Yaskawa INFORM job: v1_150 (2).JBI

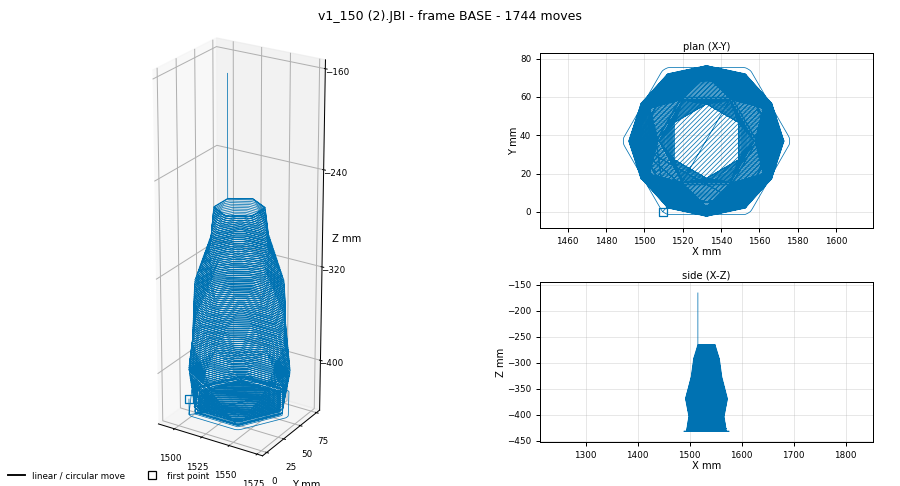
[picture p0: tool path of v1_150 (2).JBI in frame BASE, 1744 of 1745 moves have a stored position in this frame; points joined in program order, loops and branches not executed]
/JOB
//NAME v1_150
//POS
///NPOS 1745,0,0,0,0,0
///TOOL 10
///POSTYPE PULSE
///PULSE
C00000=0,15,42,180,57,90
///TOOL 10
///POSTYPE BASE
///RECTAN
///RCONF 0,0,0,0,0,0,0,0
C00001=1509.595,0.130,-417.872,180.00,-0.00,0.00
C00002=1509.595,0.130,-431.372,-180.00,-0.00,0.00
C00003=1510.195,-0.324,-431.372,180.00,-0.00,0.00
C00004=1510.690,-0.621,-431.372,180.00,-0.00,0.00
C00005=1511.242,-0.928,-431.372,180.00,-0.00,0.00
C00006=1511.746,-1.163,-431.372,-180.00,-0.00,0.00
C00007=1512.279,-1.323,-431.372,-180.00,-0.00,0.00
C00008=1513.047,-1.416,-431.372,-180.00,-0.00,0.00
C00009=1514.162,-1.438,-431.372,180.00,-0.00,0.00
C00010=1551.066,-1.438,-431.372,180.00,-0.00,0.00
C00011=1551.770,-1.428,-431.372,180.00,-0.00,0.00
C00012=1552.324,-1.380,-431.372,-180.00,-0.00,0.00
C00013=1552.866,-1.253,-431.372,-180.00,-0.00,0.00
C00014=1553.563,-0.959,-431.372,180.00,-0.00,0.00
C00015=1554.028,-0.703,-431.372,-180.00,-0.00,0.00
C00016=1554.602,-0.361,-431.372,-180.00,-0.00,0.00
C00017=1555.059,-0.043,-431.372,-180.00,-0.00,0.00
C00018=1555.465,0.338,-431.372,-180.00,-0.00,0.00
C00019=1555.933,0.960,-431.372,-180.00,-0.00,0.00
C00020=1556.527,1.941,-431.372,180.00,-0.00,0.00
///RCONF 0,0,0,1,0,0,0,0
C00021=1574.971,33.887,-431.372,180.00,-0.00,0.00
C00022=1575.305,34.482,-431.372,180.00,-0.00,0.00
C00023=1575.542,34.986,-431.372,180.00,-0.00,0.00
C00024=1575.704,35.518,-431.372,180.00,-0.00,0.00
C00025=1575.800,36.272,-431.372,180.00,-0.00,0.00
C00026=1575.812,36.838,-431.372,180.00,-0.00,0.00
C00027=1575.802,37.485,-431.372,180.00,-0.00,0.00
C00028=1575.753,38.039,-431.372,180.00,-0.00,0.00
C00029=1575.626,38.581,-431.372,-180.00,-0.00,0.00
C00030=1575.323,39.291,-431.372,-180.00,-0.00,0.00
C00031=1574.749,40.335,-431.372,-180.00,-0.00,0.00
C00032=1556.343,72.213,-431.372,180.00,-0.00,0.00
C00033=1555.982,72.818,-431.372,-180.00,-0.00,0.00
C00034=1555.663,73.274,-431.372,-180.00,-0.00,0.00
C00035=1555.282,73.679,-431.372,180.00,-0.00,0.00
C00036=1554.663,74.145,-431.372,-180.00,-0.00,0.00
C00037=1553.870,74.624,-431.372,180.00,-0.00,0.00
C00038=1553.416,74.870,-431.372,-180.00,-0.00,0.00
C00039=1553.391,74.882,-431.372,180.00,-0.00,0.00
C00040=1552.873,75.087,-431.372,180.00,-0.00,0.00
C00041=1552.332,75.214,-431.372,180.00,-0.00,0.00
C00042=1551.828,75.262,-431.372,-180.00,-0.00,0.00
C00043=1551.375,75.274,-431.372,180.00,-0.00,0.00
C00044=1513.794,75.274,-431.372,180.00,-0.00,0.00
C00045=1513.090,75.264,-431.372,-180.00,-0.00,0.00
C00046=1512.536,75.216,-431.372,180.00,-0.00,0.00
C00047=1511.994,75.089,-431.372,180.00,-0.00,0.00
C00048=1511.295,74.794,-431.372,180.00,-0.00,0.00
C00049=1510.814,74.529,-431.372,180.00,-0.00,0.00
C00050=1510.254,74.195,-431.372,-180.00,-0.00,0.00
C00051=1509.798,73.876,-431.372,-180.00,-0.00,0.00
C00052=1509.392,73.496,-431.372,-180.00,-0.00,0.00
C00053=1508.921,72.869,-431.372,-180.00,-0.00,0.00
C00054=1508.309,71.854,-431.372,180.00,-0.00,0.00
C00055=1489.889,39.948,-431.372,-180.00,-0.00,0.00
C00056=1489.554,39.351,-431.372,-180.00,-0.00,0.00
C00057=1489.317,38.848,-431.372,-180.00,-0.00,0.00
C00058=1489.155,38.315,-431.372,180.00,-0.00,0.00
C00059=1489.059,37.553,-431.372,180.00,-0.00,0.00
C00060=1489.048,36.998,-431.372,180.00,-0.00,0.00
C00061=1489.058,36.351,-431.372,180.00,-0.00,0.00
C00062=1489.107,35.797,-431.372,180.00,-0.00,0.00
C00063=1489.234,35.255,-431.372,-180.00,-0.00,0.00
C00064=1489.537,34.545,-431.372,180.00,-0.00,0.00
C00065=1490.111,33.501,-431.372,180.00,-0.00,0.00
///RCONF 0,0,0,0,0,0,0,0
C00066=1508.511,1.634,-431.372,180.00,-0.00,0.00
C00067=1508.895,0.991,-431.372,-180.00,-0.00,0.00
C00068=1509.214,0.535,-431.372,180.00,-0.00,0.00
C00069=1509.595,0.130,-431.372,-180.00,-0.00,0.00
///RCONF 0,0,0,1,0,0,0,0
C00070=1512.867,3.628,-431.372,180.00,-0.00,0.00
C00071=1551.455,70.424,-431.372,-180.00,-0.00,0.00
C00072=1551.482,70.524,-431.372,180.00,-0.00,0.00
C00073=1513.378,70.524,-431.372,-180.00,-0.00,0.00
C00074=1512.852,70.220,-431.372,180.00,-0.00,0.00
C00075=1493.798,37.220,-431.372,-180.00,-0.00,0.00
C00076=1493.799,36.615,-431.372,180.00,-0.00,0.00
C00077=1512.853,3.614,-431.372,180.00,-0.00,0.00
C00078=1513.378,3.312,-431.372,-180.00,-0.00,0.00
C00079=1551.482,3.312,-431.372,180.00,-0.00,0.00
C00080=1552.008,3.616,-431.372,-180.00,-0.00,0.00
C00081=1571.062,36.616,-431.372,-180.00,-0.00,0.00
C00082=1571.061,37.221,-431.372,180.00,-0.00,0.00
C00083=1552.008,70.220,-431.372,180.00,-0.00,0.00
C00084=1551.482,70.524,-431.372,180.00,-0.00,0.00
C00085=1550.607,70.524,-431.372,180.00,-0.00,0.00
C00086=1550.607,70.424,-431.372,180.00,-0.00,0.00
C00087=1550.827,68.784,-431.372,180.00,-0.00,0.00
C00088=1514.033,68.784,-431.372,180.00,-0.00,0.00
C00089=1495.634,36.919,-431.372,180.00,-0.00,0.00
C00090=1514.032,5.052,-431.372,180.00,-0.00,0.00
C00091=1550.827,5.052,-431.372,180.00,-0.00,0.00
C00092=1569.226,36.917,-431.372,-180.00,-0.00,0.00
C00093=1550.827,68.784,-431.372,180.00,-0.00,0.00
C00094=1516.485,67.996,-431.372,180.00,-0.00,0.00
C00095=1511.757,63.268,-431.372,-180.00,-0.00,0.00
C00096=1511.448,62.959,-431.372,-180.00,-0.00,0.00
C00097=1508.376,57.412,-431.372,180.00,-0.00,0.00
C00098=1518.960,67.996,-431.372,180.00,-0.00,0.00
C00099=1521.435,67.996,-431.372,180.00,-0.00,0.00
C00100=1504.995,51.555,-431.372,-180.00,-0.00,0.00
C00101=1504.686,51.246,-431.372,-180.00,-0.00,0.00
C00102=1501.614,45.700,-431.372,180.00,-0.00,0.00
C00103=1523.910,67.996,-431.372,-180.00,-0.00,0.00
C00104=1526.385,67.996,-431.372,-180.00,-0.00,0.00
C00105=1498.233,39.844,-431.372,180.00,-0.00,0.00
C00106=1497.924,39.535,-431.372,-180.00,-0.00,0.00
C00107=1496.995,36.131,-431.372,-180.00,-0.00,0.00
C00108=1528.859,67.996,-431.372,-180.00,-0.00,0.00
C00109=1531.334,67.996,-431.372,-180.00,-0.00,0.00
C00110=1497.901,34.562,-431.372,180.00,-0.00,0.00
C00111=1498.807,32.993,-431.372,-180.00,-0.00,0.00
C00112=1533.809,67.996,-431.372,-180.00,-0.00,0.00
C00113=1536.284,67.996,-431.372,180.00,-0.00,0.00
C00114=1499.713,31.424,-431.372,-180.00,-0.00,0.00
C00115=1500.618,29.855,-431.372,180.00,-0.00,0.00
C00116=1538.759,67.996,-431.372,-180.00,-0.00,0.00
C00117=1541.234,67.996,-431.372,180.00,-0.00,0.00
C00118=1501.524,28.286,-431.372,-180.00,-0.00,0.00
C00119=1502.430,26.717,-431.372,180.00,-0.00,0.00
C00120=1543.709,67.996,-431.372,180.00,-0.00,0.00
C00121=1546.184,67.996,-431.372,180.00,-0.00,0.00
C00122=1503.336,25.149,-431.372,180.00,-0.00,0.00
C00123=1504.242,23.579,-431.372,180.00,-0.00,0.00
C00124=1548.658,67.996,-431.372,-180.00,-0.00,0.00
C00125=1550.650,67.513,-431.372,180.00,-0.00,0.00
C00126=1505.148,22.010,-431.372,180.00,-0.00,0.00
C00127=1506.054,20.441,-431.372,180.00,-0.00,0.00
C00128=1551.556,65.944,-431.372,180.00,-0.00,0.00
C00129=1552.462,64.375,-431.372,180.00,-0.00,0.00
C00130=1506.960,18.872,-431.372,-180.00,-0.00,0.00
C00131=1507.865,17.303,-431.372,-180.00,-0.00,0.00
C00132=1553.369,62.806,-431.372,-180.00,-0.00,0.00
C00133=1554.274,61.237,-431.372,180.00,-0.00,0.00
C00134=1508.771,15.734,-431.372,180.00,-0.00,0.00
C00135=1509.677,14.165,-431.372,-180.00,-0.00,0.00
C00136=1555.180,59.668,-431.372,-180.00,-0.00,0.00
C00137=1556.086,58.099,-431.372,180.00,-0.00,0.00
C00138=1510.583,12.596,-431.372,180.00,-0.00,0.00
C00139=1511.489,11.027,-431.372,-180.00,-0.00,0.00
C00140=1556.992,56.530,-431.372,-180.00,-0.00,0.00
C00141=1557.898,54.961,-431.372,180.00,-0.00,0.00
C00142=1512.394,9.458,-431.372,-180.00,-0.00,0.00
C00143=1513.300,7.889,-431.372,-180.00,-0.00,0.00
C00144=1558.804,53.393,-431.372,-180.00,-0.00,0.00
C00145=1559.710,51.823,-431.372,180.00,-0.00,0.00
C00146=1514.206,6.320,-431.372,-180.00,-0.00,0.00
C00147=1516.200,5.839,-431.372,-180.00,-0.00,0.00
C00148=1560.616,50.254,-431.372,-180.00,-0.00,0.00
C00149=1561.521,48.685,-431.372,-180.00,-0.00,0.00
C00150=1518.675,5.839,-431.372,-180.00,-0.00,0.00
C00151=1521.150,5.839,-431.372,-180.00,-0.00,0.00
C00152=1562.427,47.116,-431.372,180.00,-0.00,0.00
C00153=1563.333,45.547,-431.372,180.00,-0.00,0.00
C00154=1523.625,5.839,-431.372,-180.00,-0.00,0.00
C00155=1526.100,5.839,-431.372,-180.00,-0.00,0.00
C00156=1564.240,43.979,-431.372,180.00,-0.00,0.00
C00157=1565.145,42.410,-431.372,180.00,-0.00,0.00
C00158=1528.575,5.839,-431.372,-180.00,-0.00,0.00
C00159=1531.049,5.839,-431.372,-180.00,-0.00,0.00
C00160=1566.051,40.841,-431.372,-180.00,-0.00,0.00
C00161=1566.957,39.272,-431.372,180.00,-0.00,0.00
C00162=1533.524,5.839,-431.372,180.00,-0.00,0.00
C00163=1535.999,5.839,-431.372,-180.00,-0.00,0.00
C00164=1567.863,37.703,-431.372,-180.00,-0.00,0.00
C00165=1568.172,38.012,-431.372,180.00,-0.00,0.00
C00166=1566.627,33.992,-431.372,-180.00,-0.00,0.00
C00167=1538.474,5.839,-431.372,-180.00,-0.00,0.00
C00168=1540.949,5.839,-431.372,-180.00,-0.00,0.00
C00169=1563.246,28.136,-431.372,-180.00,-0.00,0.00
C00170=1563.555,28.445,-431.372,180.00,-0.00,0.00
C00171=1559.865,22.280,-431.372,180.00,-0.00,0.00
C00172=1543.424,5.839,-431.372,180.00,-0.00,0.00
C00173=1545.899,5.839,-431.372,180.00,-0.00,0.00
C00174=1556.483,16.424,-431.372,180.00,-0.00,0.00
C00175=1556.792,16.733,-431.372,180.00,-0.00,0.00
C00176=1553.102,10.567,-431.372,-180.00,-0.00,0.00
C00177=1548.373,5.839,-431.372,180.00,-0.00,0.00
C00178=1548.064,5.530,-431.372,-180.00,-0.00,0.00
C00179=1548.064,5.530,-429.872,-180.00,-0.00,0.00
C00180=1494.414,35.749,-429.872,-180.00,-0.00,0.00
C00181=1494.043,35.534,-429.872,180.00,-0.00,0.00
C00182=1512.039,4.366,-429.872,180.00,-0.00,0.00
C00183=1514.436,2.983,-429.872,180.00,-0.00,0.00
C00184=1550.425,2.983,-429.872,180.00,-0.00,0.00
C00185=1552.822,4.368,-429.872,180.00,-0.00,0.00
C00186=1570.817,35.535,-429.872,-180.00,-0.00,0.00
C00187=1570.817,38.302,-429.872,-180.00,-0.00,0.00
C00188=1552.821,69.470,-429.872,-180.00,-0.00,0.00
C00189=1550.424,70.853,-429.872,180.00,-0.00,0.00
C00190=1514.435,70.853,-429.872,180.00,-0.00,0.00
C00191=1512.038,69.468,-429.872,-180.00,-0.00,0.00
C00192=1494.043,38.301,-429.872,180.00,-0.00,0.00
C00193=1494.043,35.534,-429.872,180.00,-0.00,0.00
C00194=1493.799,36.615,-429.872,180.00,-0.00,0.00
C00195=1512.278,4.505,-429.633,-180.00,-0.00,0.00
C00196=1514.436,3.256,-429.617,180.00,-0.00,0.00
C00197=1550.425,3.206,-429.385,180.00,-0.00,0.00
C00198=1552.632,4.477,-429.369,180.00,-0.00,0.00
C00199=1570.671,35.619,-429.137,-180.00,-0.00,0.00
C00200=1570.675,38.219,-429.120,-180.00,-0.00,0.00
C00201=1552.723,69.413,-428.888,-180.00,-0.00,0.00
C00202=1550.424,70.743,-428.871,180.00,-0.00,0.00
C00203=1514.435,70.794,-428.639,-180.00,-0.00,0.00
C00204=1512.086,69.440,-428.622,-180.00,-0.00,0.00
C00205=1494.047,38.299,-428.390,-180.00,-0.00,0.00
C00206=1494.043,35.534,-428.372,-180.00,-0.00,0.00
C00207=1519.293,14.162,-428.070,-180.00,-0.00,0.00
C00208=1545.567,14.162,-427.831,180.00,-0.00,0.00
C00209=1558.706,36.918,-427.591,180.00,-0.00,0.00
C00210=1545.567,59.674,-427.351,180.00,-0.00,0.00
C00211=1519.293,59.674,-427.112,-180.00,-0.00,0.00
C00212=1506.154,36.918,-426.872,180.00,-0.00,0.00
C00213=1506.266,36.912,-426.872,180.00,-0.00,0.00
C00214=1519.303,59.657,-426.872,-180.00,-0.00,0.00
C00215=1517.955,60.437,-426.872,180.00,-0.00,0.00
C00216=1512.921,63.340,-426.872,180.00,-0.00,0.00
C00217=1511.588,64.111,-426.872,-180.00,-0.00,0.00
C00218=1513.794,68.122,-426.872,-180.00,-0.00,0.00
C00219=1513.864,68.052,-426.872,-180.00,-0.00,0.00
C00220=1514.750,68.563,-426.872,-180.00,-0.00,0.00
C00221=1550.109,68.564,-426.872,-180.00,-0.00,0.00
C00222=1550.995,68.053,-426.872,-180.00,-0.00,0.00
C00223=1568.676,37.431,-426.872,180.00,-0.00,0.00
C00224=1568.677,36.407,-426.872,-180.00,-0.00,0.00
C00225=1550.996,5.784,-426.872,180.00,-0.00,0.00
C00226=1550.110,5.273,-426.872,-180.00,-0.00,0.00
C00227=1514.751,5.272,-426.872,180.00,-0.00,0.00
C00228=1513.865,5.783,-426.872,-180.00,-0.00,0.00
C00229=1496.184,36.405,-426.872,-180.00,-0.00,0.00
C00230=1496.183,37.429,-426.872,-180.00,-0.00,0.00
C00231=1513.864,68.052,-426.872,-180.00,-0.00,0.00
C00232=1514.622,68.489,-426.872,-180.00,-0.00,0.00
C00233=1514.571,68.575,-426.872,-180.00,-0.00,0.00
C00234=1549.340,71.086,-426.872,-180.00,-0.00,0.00
C00235=1549.365,71.182,-426.872,180.00,-0.00,0.00
C00236=1515.494,71.182,-426.872,-180.00,-0.00,0.00
C00237=1511.223,68.715,-426.872,180.00,-0.00,0.00
C00238=1494.287,39.382,-426.872,-180.00,-0.00,0.00
C00239=1494.288,34.451,-426.872,180.00,-0.00,0.00
C00240=1511.225,5.118,-426.872,-180.00,-0.00,0.00
C00241=1515.495,2.654,-426.872,180.00,-0.00,0.00
C00242=1549.366,2.654,-426.872,-180.00,-0.00,0.00
C00243=1553.637,5.121,-426.872,-180.00,-0.00,0.00
C00244=1570.573,34.454,-426.872,180.00,-0.00,0.00
C00245=1570.572,39.385,-426.872,180.00,-0.00,0.00
C00246=1553.635,68.718,-426.872,-180.00,-0.00,0.00
C00247=1549.365,71.182,-426.872,180.00,-0.00,0.00
C00248=1548.490,71.182,-426.872,-180.00,-0.00,0.00
C00249=1548.490,71.082,-426.872,-180.00,-0.00,0.00
C00250=1514.750,68.563,-426.872,-180.00,-0.00,0.00
C00251=1515.160,67.025,-426.872,-180.00,-0.00,0.00
C00252=1519.303,61.214,-426.872,180.00,-0.00,0.00
C00253=1519.303,59.657,-426.872,-180.00,-0.00,0.00
C00254=1506.266,36.912,-426.872,180.00,-0.00,0.00
C00255=1506.154,36.918,-426.872,180.00,-0.00,0.00
C00256=1510.409,5.871,-426.670,-180.00,-0.00,0.00
///RCONF 0,0,0,0,0,0,0,0
C00257=1516.555,2.324,-426.624,180.00,-0.00,0.00
C00258=1548.305,2.324,-426.420,180.00,-0.00,0.00
///RCONF 0,0,0,1,0,0,0,0
C00259=1554.452,5.872,-426.374,180.00,-0.00,0.00
C00260=1570.328,33.372,-426.169,-180.00,-0.00,0.00
C00261=1570.327,40.467,-426.123,180.00,-0.00,0.00
C00262=1554.450,67.965,-425.919,180.00,-0.00,0.00
C00263=1548.305,71.512,-425.873,-180.00,-0.00,0.00
C00264=1516.555,71.512,-425.668,180.00,-0.00,0.00
C00265=1510.408,67.964,-425.622,-180.00,-0.00,0.00
C00266=1494.532,40.464,-425.418,180.00,-0.00,0.00
C00267=1494.533,33.369,-425.372,-180.00,-0.00,0.00
C00268=1509.843,6.766,-425.175,180.00,-0.00,0.00
///RCONF 0,0,0,0,0,0,0,0
C00269=1517.615,2.268,-425.117,-180.00,-0.00,0.00
C00270=1547.247,2.227,-424.927,-180.00,-0.00,0.00
///RCONF 0,0,0,1,0,0,0,0
C00271=1555.078,6.736,-424.869,180.00,-0.00,0.00
C00272=1569.930,32.380,-424.679,-180.00,-0.00,0.00
C00273=1569.942,41.464,-424.620,180.00,-0.00,0.00
C00274=1555.159,67.150,-424.430,-180.00,-0.00,0.00
C00275=1547.245,71.731,-424.371,180.00,-0.00,0.00
C00276=1517.613,71.773,-424.181,-180.00,-0.00,0.00
C00277=1509.640,67.181,-424.122,180.00,-0.00,0.00
C00278=1494.788,41.539,-423.931,-180.00,-0.00,0.00
C00279=1494.776,32.289,-423.872,180.00,-0.00,0.00
C00280=1509.032,7.522,-423.689,180.00,-0.00,0.00
///RCONF 0,0,0,0,0,0,0,0
C00281=1518.674,1.939,-423.617,180.00,-0.00,0.00
C00282=1546.188,1.901,-423.441,180.00,-0.00,0.00
///RCONF 0,0,0,1,0,0,0,0
C00283=1555.893,7.489,-423.369,-180.00,-0.00,0.00
C00284=1569.682,31.298,-423.192,-180.00,-0.00,0.00
C00285=1569.697,42.546,-423.120,-180.00,-0.00,0.00
C00286=1555.971,66.397,-422.944,-180.00,-0.00,0.00
C00287=1546.186,72.060,-422.871,180.00,-0.00,0.00
C00288=1518.672,72.099,-422.695,180.00,-0.00,0.00
C00289=1508.825,66.428,-422.622,180.00,-0.00,0.00
C00290=1495.035,42.618,-422.445,180.00,-0.00,0.00
C00291=1495.021,31.207,-422.372,180.00,-0.00,0.00
C00292=1508.218,8.276,-422.202,180.00,-0.00,0.00
///RCONF 0,0,0,0,0,0,0,0
C00293=1519.730,1.610,-422.117,180.00,-0.00,0.00
C00294=1545.130,1.575,-421.954,180.00,-0.00,0.00
///RCONF 0,0,0,1,0,0,0,0
C00295=1556.705,8.239,-421.869,180.00,-0.00,0.00
C00296=1569.436,30.219,-421.706,-180.00,-0.00,0.00
C00297=1569.452,43.627,-421.620,180.00,-0.00,0.00
C00298=1556.783,65.642,-421.457,180.00,-0.00,0.00
C00299=1545.130,72.389,-421.371,-180.00,-0.00,0.00
C00300=1519.730,72.425,-421.208,-180.00,-0.00,0.00
C00301=1508.013,65.679,-421.122,180.00,-0.00,0.00
C00302=1495.282,43.699,-420.959,180.00,-0.00,0.00
C00303=1495.266,30.126,-420.872,180.00,-0.00,0.00
C00304=1507.406,9.031,-420.716,-180.00,-0.00,0.00
///RCONF 0,0,0,0,0,0,0,0
C00305=1520.790,1.281,-420.617,-180.00,-0.00,0.00
C00306=1544.070,1.249,-420.468,-180.00,-0.00,0.00
///RCONF 0,0,0,1,0,0,0,0
C00307=1557.520,8.992,-420.369,180.00,-0.00,0.00
C00308=1569.189,29.140,-420.220,-180.00,-0.00,0.00
C00309=1569.208,44.709,-420.120,-180.00,-0.00,0.00
C00310=1557.595,64.887,-419.971,-180.00,-0.00,0.00
C00311=1544.070,72.718,-419.871,180.00,-0.00,0.00
C00312=1520.790,72.751,-419.722,180.00,-0.00,0.00
C00313=1507.199,64.925,-419.622,-180.00,-0.00,0.00
C00314=1495.530,44.781,-419.473,180.00,-0.00,0.00
C00315=1495.510,29.044,-419.372,180.00,-0.00,0.00
C00316=1506.595,9.785,-419.230,-180.00,-0.00,0.00
///RCONF 0,0,0,0,0,0,0,0
C00317=1521.848,0.952,-419.117,180.00,-0.00,0.00
C00318=1543.012,0.923,-418.982,-180.00,-0.00,0.00
///RCONF 0,0,0,1,0,0,0,0
C00319=1558.334,9.744,-418.869,-180.00,-0.00,0.00
C00320=1568.940,28.059,-418.734,180.00,-0.00,0.00
C00321=1568.963,45.792,-418.620,180.00,-0.00,0.00
C00322=1558.407,64.133,-418.485,180.00,-0.00,0.00
C00323=1543.012,73.047,-418.371,-180.00,-0.00,0.00
C00324=1521.848,73.077,-418.236,180.00,-0.00,0.00
C00325=1506.384,64.173,-418.122,180.00,-0.00,0.00
C00326=1495.777,45.861,-417.986,-180.00,-0.00,0.00
C00327=1495.755,27.961,-417.872,180.00,-0.00,0.00
C00328=1505.782,10.538,-417.744,180.00,-0.00,0.00
///RCONF 0,0,0,0,0,0,0,0
C00329=1522.907,0.623,-417.617,-180.00,-0.00,0.00
C00330=1541.953,0.597,-417.496,-180.00,-0.00,0.00
///RCONF 0,0,0,1,0,0,0,0
C00331=1559.148,10.496,-417.369,180.00,-0.00,0.00
C00332=1568.693,26.977,-417.247,180.00,-0.00,0.00
C00333=1568.719,46.873,-417.120,-180.00,-0.00,0.00
C00334=1559.219,63.380,-416.999,180.00,-0.00,0.00
C00335=1541.953,73.376,-416.871,180.00,-0.00,0.00
C00336=1522.907,73.403,-416.750,-180.00,-0.00,0.00
C00337=1505.570,63.421,-416.622,-180.00,-0.00,0.00
C00338=1496.024,46.942,-416.500,180.00,-0.00,0.00
C00339=1495.999,26.880,-416.372,180.00,-0.00,0.00
C00340=1504.971,11.292,-416.257,-180.00,-0.00,0.00
///RCONF 0,0,0,0,0,0,0,0
C00341=1523.967,0.294,-416.117,180.00,-0.00,0.00
C00342=1540.889,0.270,-416.009,-180.00,-0.00,0.00
///RCONF 0,0,0,1,0,0,0,0
C00343=1559.963,11.249,-415.869,-180.00,-0.00,0.00
C00344=1568.447,25.896,-415.761,180.00,-0.00,0.00
C00345=1568.474,47.955,-415.620,180.00,-0.00,0.00
C00346=1560.031,62.626,-415.512,-180.00,-0.00,0.00
C00347=1540.893,73.705,-415.371,-180.00,-0.00,0.00
C00348=1523.971,73.730,-415.263,-180.00,-0.00,0.00
C00349=1504.755,62.668,-415.122,180.00,-0.00,0.00
C00350=1496.271,48.022,-415.014,-180.00,-0.00,0.00
C00351=1496.244,25.798,-414.872,-180.00,-0.00,0.00
C00352=1504.158,12.046,-414.771,180.00,-0.00,0.00
///RCONF 0,0,0,0,0,0,0,0
C00353=1525.026,-0.035,-414.617,180.00,-0.00,0.00
C00354=1539.831,-0.056,-414.523,-180.00,-0.00,0.00
///RCONF 0,0,0,1,0,0,0,0
C00355=1560.777,12.001,-414.369,-180.00,-0.00,0.00
C00356=1568.200,24.816,-414.275,-180.00,-0.00,0.00
C00357=1568.230,49.036,-414.120,180.00,-0.00,0.00
C00358=1560.843,61.872,-414.026,-180.00,-0.00,0.00
C00359=1539.834,74.034,-413.871,-180.00,-0.00,0.00
C00360=1525.029,74.057,-413.777,-180.00,-0.00,0.00
C00361=1503.941,61.916,-413.622,180.00,-0.00,0.00
C00362=1496.518,49.102,-413.527,180.00,-0.00,0.00
C00363=1496.488,24.717,-413.372,-180.00,-0.00,0.00
C00364=1503.347,12.801,-413.284,-180.00,-0.00,0.00
///RCONF 0,0,0,0,0,0,0,0
C00365=1526.085,-0.364,-413.117,180.00,-0.00,0.00
C00366=1538.773,-0.382,-413.036,-180.00,-0.00,0.00
///RCONF 0,0,0,1,0,0,0,0
C00367=1561.592,12.754,-412.869,180.00,-0.00,0.00
C00368=1567.953,23.736,-412.788,180.00,-0.00,0.00
C00369=1567.985,50.118,-412.620,180.00,-0.00,0.00
C00370=1561.655,61.117,-412.539,-180.00,-0.00,0.00
C00371=1538.775,74.363,-412.371,180.00,-0.00,0.00
C00372=1526.087,74.383,-412.290,-180.00,-0.00,0.00
C00373=1503.126,61.163,-412.122,180.00,-0.00,0.00
C00374=1496.766,50.182,-412.041,-180.00,-0.00,0.00
C00375=1496.733,23.635,-411.872,180.00,-0.00,0.00
C00376=1502.535,13.554,-411.798,-180.00,-0.00,0.00
///RCONF 0,0,0,0,0,0,0,0
C00377=1527.144,-0.693,-411.617,-180.00,-0.00,0.00
C00378=1537.712,-0.708,-411.550,-180.00,-0.00,0.00
///RCONF 0,0,0,1,0,0,0,0
C00379=1562.406,13.507,-411.369,180.00,-0.00,0.00
C00380=1567.706,22.658,-411.302,180.00,-0.00,0.00
C00381=1567.740,51.200,-411.120,-180.00,-0.00,0.00
C00382=1562.467,60.364,-411.053,180.00,-0.00,0.00
C00383=1537.716,74.692,-410.871,180.00,-0.00,0.00
C00384=1527.148,74.709,-410.804,180.00,-0.00,0.00
C00385=1502.312,60.411,-410.622,-180.00,-0.00,0.00
C00386=1497.012,51.263,-410.555,180.00,-0.00,0.00
C00387=1496.978,22.553,-410.372,180.00,-0.00,0.00
C00388=1501.722,14.310,-410.312,-180.00,-0.00,0.00
///RCONF 0,0,0,0,0,0,0,0
C00389=1528.203,-1.022,-410.117,180.00,-0.00,0.00
C00390=1536.657,-1.034,-410.064,-180.00,-0.00,0.00
///RCONF 0,0,0,1,0,0,0,0
C00391=1563.221,14.259,-409.869,180.00,-0.00,0.00
C00392=1567.458,21.576,-409.815,180.00,-0.00,0.00
C00393=1567.496,52.282,-409.620,180.00,-0.00,0.00
C00394=1563.279,59.608,-409.567,180.00,-0.00,0.00
C00395=1536.657,75.022,-409.371,-180.00,-0.00,0.00
C00396=1528.203,75.034,-409.317,-180.00,-0.00,0.00
C00397=1501.497,59.657,-409.122,180.00,-0.00,0.00
C00398=1497.260,52.343,-409.068,180.00,-0.00,0.00
C00399=1497.222,21.471,-408.872,-180.00,-0.00,0.00
C00400=1500.911,15.063,-408.825,-180.00,-0.00,0.00
///RCONF 0,0,0,0,0,0,0,0
C00401=1529.262,-1.352,-408.617,180.00,-0.00,0.00
C00402=1535.598,-1.360,-408.577,180.00,-0.00,0.00
///RCONF 0,0,0,1,0,0,0,0
C00403=1564.035,15.011,-408.369,-180.00,-0.00,0.00
C00404=1567.211,20.497,-408.329,180.00,-0.00,0.00
C00405=1567.251,53.364,-408.120,-180.00,-0.00,0.00
C00406=1564.091,58.855,-408.080,-180.00,-0.00,0.00
C00407=1535.598,75.351,-407.871,180.00,-0.00,0.00
C00408=1529.262,75.360,-407.831,-180.00,-0.00,0.00
C00409=1500.683,58.906,-407.622,-180.00,-0.00,0.00
C00410=1497.506,53.423,-407.582,180.00,-0.00,0.00
C00411=1497.467,20.389,-407.372,180.00,-0.00,0.00
C00412=1500.098,15.817,-407.339,180.00,-0.00,0.00
///RCONF 0,0,0,0,0,0,0,0
C00413=1530.321,-1.681,-407.117,180.00,-0.00,0.00
C00414=1534.539,-1.686,-407.091,-180.00,-0.00,0.00
///RCONF 0,0,0,1,0,0,0,0
C00415=1564.850,15.764,-406.869,180.00,-0.00,0.00
C00416=1566.964,19.415,-406.842,180.00,-0.00,0.00
C00417=1567.007,54.445,-406.620,-180.00,-0.00,0.00
C00418=1564.903,58.101,-406.593,-180.00,-0.00,0.00
C00419=1534.539,75.680,-406.371,-180.00,-0.00,0.00
C00420=1530.321,75.686,-406.344,180.00,-0.00,0.00
C00421=1499.868,58.153,-406.122,-180.00,-0.00,0.00
C00422=1497.754,54.503,-406.095,-180.00,-0.00,0.00
C00423=1497.711,19.308,-405.872,180.00,-0.00,0.00
C00424=1499.287,16.571,-405.852,180.00,-0.00,0.00
///RCONF 0,0,0,0,0,0,0,0
C00425=1531.380,-2.010,-405.617,-180.00,-0.00,0.00
C00426=1533.480,-2.012,-405.604,180.00,-0.00,0.00
///RCONF 0,0,0,1,0,0,0,0
C00427=1565.665,16.517,-405.369,-180.00,-0.00,0.00
C00428=1566.718,18.336,-405.356,180.00,-0.00,0.00
C00429=1566.762,55.528,-405.120,-180.00,-0.00,0.00
C00430=1565.715,57.347,-405.107,180.00,-0.00,0.00
C00431=1533.480,76.009,-404.871,-180.00,-0.00,0.00
C00432=1531.380,76.012,-404.858,180.00,-0.00,0.00
C00433=1499.053,57.400,-404.622,180.00,-0.00,0.00
C00434=1498.000,55.582,-404.608,-180.00,-0.00,0.00
C00435=1497.956,18.225,-404.372,180.00,-0.00,0.00
///RCONF 0,0,0,0,0,0,0,0
C00436=1532.430,-2.337,-404.118,-180.00,-0.00,0.00
///RCONF 0,0,0,1,0,0,0,0
C00437=1566.473,17.262,-403.870,180.00,-0.00,0.00
C00438=1566.520,56.600,-403.621,180.00,-0.00,0.00
C00439=1532.430,76.335,-403.371,-180.00,-0.00,0.00
C00440=1498.247,56.654,-403.122,180.00,-0.00,0.00
C00441=1498.200,17.155,-402.872,-180.00,-0.00,0.00
C00442=1498.701,16.866,-402.868,-180.00,-0.00,0.00
///RCONF 0,0,0,0,0,0,0,0
C00443=1531.912,-2.345,-402.625,-180.00,-0.00,0.00
C00444=1532.946,-2.348,-402.618,-180.00,-0.00,0.00
///RCONF 0,0,0,1,0,0,0,0
C00445=1566.189,16.806,-402.375,-180.00,-0.00,0.00
C00446=1566.728,17.735,-402.368,180.00,-0.00,0.00
C00447=1566.761,56.103,-402.124,-180.00,-0.00,0.00
C00448=1566.210,57.059,-402.117,180.00,-0.00,0.00
C00449=1532.999,76.270,-401.874,180.00,-0.00,0.00
C00450=1531.863,76.273,-401.867,180.00,-0.00,0.00
C00451=1498.620,57.118,-401.623,180.00,-0.00,0.00
C00452=1498.030,56.101,-401.616,-180.00,-0.00,0.00
C00453=1497.997,17.732,-401.372,-180.00,-0.00,0.00
C00454=1499.367,16.243,-401.359,-180.00,-0.00,0.00
///RCONF 0,0,0,0,0,0,0,0
C00455=1531.037,-2.090,-401.127,180.00,-0.00,0.00
C00456=1533.826,-2.093,-401.109,180.00,-0.00,0.00
///RCONF 0,0,0,1,0,0,0,0
C00457=1565.541,16.165,-400.876,-180.00,-0.00,0.00
C00458=1566.961,18.619,-400.858,180.00,-0.00,0.00
C00459=1567.005,55.219,-400.626,-180.00,-0.00,0.00
C00460=1565.566,57.716,-400.607,-180.00,-0.00,0.00
C00461=1533.895,76.052,-400.375,180.00,-0.00,0.00
C00462=1530.962,76.054,-400.356,-180.00,-0.00,0.00
C00463=1499.247,57.795,-400.124,180.00,-0.00,0.00
C00464=1497.755,55.217,-400.105,180.00,-0.00,0.00
C00465=1497.711,18.619,-399.872,180.00,-0.00,0.00
C00466=1499.988,15.552,-399.848,-180.00,-0.00,0.00
///RCONF 0,0,0,0,0,0,0,0
C00467=1530.127,-1.897,-399.627,180.00,-0.00,0.00
C00468=1534.738,-1.900,-399.597,180.00,-0.00,0.00
///RCONF 0,0,0,1,0,0,0,0
C00469=1564.918,15.475,-399.376,180.00,-0.00,0.00
C00470=1567.250,19.504,-399.347,-180.00,-0.00,0.00
C00471=1567.292,54.331,-399.126,180.00,-0.00,0.00
C00472=1564.944,58.409,-399.096,-180.00,-0.00,0.00
C00473=1534.805,75.858,-398.875,-180.00,-0.00,0.00
C00474=1530.050,75.861,-398.845,-180.00,-0.00,0.00
C00475=1499.870,58.485,-398.624,180.00,-0.00,0.00
C00476=1497.466,54.332,-398.593,-180.00,-0.00,0.00
C00477=1497.424,19.504,-398.372,-180.00,-0.00,0.00
C00478=1500.611,14.858,-398.336,180.00,-0.00,0.00
///RCONF 0,0,0,0,0,0,0,0
C00479=1529.216,-1.701,-398.127,-180.00,-0.00,0.00
C00480=1535.650,-1.708,-398.086,-180.00,-0.00,0.00
///RCONF 0,0,0,1,0,0,0,0
C00481=1564.293,14.783,-397.876,180.00,-0.00,0.00
C00482=1567.539,20.391,-397.835,-180.00,-0.00,0.00
C00483=1567.579,53.443,-397.626,180.00,-0.00,0.00
C00484=1564.320,59.103,-397.584,180.00,-0.00,0.00
C00485=1535.716,75.662,-397.375,180.00,-0.00,0.00
C00486=1529.138,75.668,-397.333,-180.00,-0.00,0.00
C00487=1500.495,59.177,-397.124,-180.00,-0.00,0.00
C00488=1497.176,53.445,-397.082,180.00,-0.00,0.00
C00489=1497.137,20.391,-396.872,180.00,-0.00,0.00
C00490=1501.234,14.167,-396.825,180.00,-0.00,0.00
///RCONF 0,0,0,0,0,0,0,0
C00491=1528.303,-1.505,-396.627,180.00,-0.00,0.00
C00492=1536.559,-1.517,-396.574,-180.00,-0.00,0.00
///RCONF 0,0,0,1,0,0,0,0
C00493=1563.669,14.092,-396.376,-180.00,-0.00,0.00
C00494=1567.828,21.277,-396.324,180.00,-0.00,0.00
C00495=1567.865,52.558,-396.126,180.00,-0.00,0.00
C00496=1563.698,59.795,-396.073,180.00,-0.00,0.00
C00497=1536.629,75.466,-395.875,-180.00,-0.00,0.00
C00498=1528.229,75.477,-395.822,-180.00,-0.00,0.00
C00499=1501.119,59.868,-395.624,180.00,-0.00,0.00
C00500=1496.888,52.559,-395.570,-180.00,-0.00,0.00
C00501=1496.851,21.277,-395.372,180.00,-0.00,0.00
C00502=1501.857,13.474,-395.313,180.00,-0.00,0.00
///RCONF 0,0,0,0,0,0,0,0
C00503=1527.395,-1.312,-395.127,180.00,-0.00,0.00
C00504=1537.472,-1.323,-395.063,180.00,-0.00,0.00
///RCONF 0,0,0,1,0,0,0,0
C00505=1563.044,13.400,-394.876,-180.00,-0.00,0.00
C00506=1568.117,22.163,-394.812,-180.00,-0.00,0.00
C00507=1568.152,51.672,-394.626,-180.00,-0.00,0.00
C00508=1563.075,60.487,-394.561,-180.00,-0.00,0.00
C00509=1537.537,75.273,-394.375,180.00,-0.00,0.00
C00510=1527.315,75.283,-394.310,-180.00,-0.00,0.00
C00511=1501.744,60.561,-394.124,-180.00,-0.00,0.00
C00512=1496.599,51.673,-394.059,180.00,-0.00,0.00
C00513=1496.564,22.163,-393.872,180.00,-0.00,0.00
C00514=1502.481,12.780,-393.802,180.00,-0.00,0.00
///RCONF 0,0,0,0,0,0,0,0
C00515=1526.483,-1.117,-393.627,-180.00,-0.00,0.00
C00516=1538.384,-1.130,-393.552,180.00,-0.00,0.00
///RCONF 0,0,0,1,0,0,0,0
C00517=1562.420,12.708,-393.376,180.00,-0.00,0.00
C00518=1568.406,23.051,-393.301,180.00,-0.00,0.00
C00519=1568.439,50.786,-393.126,-180.00,-0.00,0.00
C00520=1562.451,61.181,-393.050,-180.00,-0.00,0.00
C00521=1538.449,75.078,-392.875,-180.00,-0.00,0.00
C00522=1526.403,75.090,-392.799,-180.00,-0.00,0.00
C00523=1502.368,61.252,-392.624,-180.00,-0.00,0.00
C00524=1496.310,50.785,-392.547,-180.00,-0.00,0.00
C00525=1496.277,23.049,-392.372,180.00,-0.00,0.00
C00526=1503.104,12.087,-392.291,-180.00,-0.00,0.00
///RCONF 0,0,0,0,0,0,0,0
C00527=1525.573,-0.923,-392.127,180.00,-0.00,0.00
C00528=1539.295,-0.937,-392.040,180.00,-0.00,0.00
///RCONF 0,0,0,1,0,0,0,0
C00529=1561.797,12.018,-391.876,-180.00,-0.00,0.00
C00530=1568.695,23.935,-391.790,180.00,-0.00,0.00
C00531=1568.726,49.896,-391.626,-180.00,-0.00,0.00
C00532=1561.828,61.874,-391.539,-180.00,-0.00,0.00
C00533=1539.359,74.884,-391.375,-180.00,-0.00,0.00
C00534=1525.492,74.897,-391.287,180.00,-0.00,0.00
C00535=1502.991,61.942,-391.124,-180.00,-0.00,0.00
C00536=1496.022,49.901,-391.036,180.00,-0.00,0.00
C00537=1495.989,23.939,-390.872,180.00,-0.00,0.00
C00538=1503.727,11.394,-390.779,180.00,-0.00,0.00
///RCONF 0,0,0,0,0,0,0,0
C00539=1524.662,-0.727,-390.627,-180.00,-0.00,0.00
C00540=1540.208,-0.743,-390.529,180.00,-0.00,0.00
///RCONF 0,0,0,1,0,0,0,0
C00541=1561.171,11.326,-390.376,-180.00,-0.00,0.00
C00542=1568.983,24.825,-390.278,180.00,-0.00,0.00
C00543=1569.012,49.015,-390.126,180.00,-0.00,0.00
C00544=1561.205,62.567,-390.027,-180.00,-0.00,0.00
C00545=1540.270,74.688,-389.875,-180.00,-0.00,0.00
C00546=1524.580,74.704,-389.776,180.00,-0.00,0.00
C00547=1503.617,62.636,-389.624,-180.00,-0.00,0.00
C00548=1495.733,49.011,-389.524,-180.00,-0.00,0.00
C00549=1495.704,24.821,-389.372,-180.00,-0.00,0.00
C00550=1504.350,10.700,-389.268,-180.00,-0.00,0.00
///RCONF 0,0,0,0,0,0,0,0
C00551=1523.751,-0.532,-389.127,180.00,-0.00,0.00
C00552=1541.120,-0.550,-389.017,-180.00,-0.00,0.00
///RCONF 0,0,0,1,0,0,0,0
C00553=1560.548,10.634,-388.876,180.00,-0.00,0.00
C00554=1569.273,25.708,-388.767,180.00,-0.00,0.00
C00555=1569.299,48.127,-388.626,-180.00,-0.00,0.00
C00556=1560.582,63.261,-388.516,180.00,-0.00,0.00
C00557=1541.181,74.493,-388.375,180.00,-0.00,0.00
C00558=1523.668,74.511,-388.265,-180.00,-0.00,0.00
C00559=1504.240,63.326,-388.124,180.00,-0.00,0.00
C00560=1495.443,48.128,-388.013,180.00,-0.00,0.00
C00561=1495.417,25.708,-387.872,-180.00,-0.00,0.00
C00562=1504.972,10.007,-387.756,180.00,-0.00,0.00
///RCONF 0,0,0,0,0,0,0,0
C00563=1522.838,-0.336,-387.627,-180.00,-0.00,0.00
C00564=1542.032,-0.358,-387.506,-180.00,-0.00,0.00
///RCONF 0,0,0,1,0,0,0,0
C00565=1559.923,9.942,-387.376,-180.00,-0.00,0.00
C00566=1569.561,26.594,-387.255,-180.00,-0.00,0.00
C00567=1569.586,47.237,-387.126,180.00,-0.00,0.00
C00568=1559.959,63.954,-387.005,-180.00,-0.00,0.00
C00569=1542.094,74.297,-386.875,180.00,-0.00,0.00
C00570=1522.756,74.319,-386.753,180.00,-0.00,0.00
C00571=1504.865,64.018,-386.624,180.00,-0.00,0.00
C00572=1495.155,47.242,-386.502,180.00,-0.00,0.00
C00573=1495.129,26.598,-386.372,-180.00,-0.00,0.00
C00574=1505.595,9.313,-386.245,-180.00,-0.00,0.00
///RCONF 0,0,0,0,0,0,0,0
C00575=1521.931,-0.144,-386.127,-180.00,-0.00,0.00
C00576=1542.943,-0.166,-385.995,180.00,-0.00,0.00
///RCONF 0,0,0,1,0,0,0,0
C00577=1559.299,9.251,-385.876,180.00,-0.00,0.00
C00578=1569.850,27.482,-385.744,180.00,-0.00,0.00
C00579=1569.872,46.355,-385.626,180.00,-0.00,0.00
C00580=1559.336,64.647,-385.493,180.00,-0.00,0.00
C00581=1543.001,74.105,-385.375,-180.00,-0.00,0.00
C00582=1521.845,74.126,-385.242,180.00,-0.00,0.00
C00583=1505.491,64.710,-385.124,180.00,-0.00,0.00
C00584=1494.866,46.354,-384.990,180.00,-0.00,0.00
C00585=1494.844,27.481,-384.872,180.00,-0.00,0.00
C00586=1506.220,8.620,-384.734,180.00,-0.00,0.00
///RCONF 0,0,0,0,0,0,0,0
C00587=1521.019,0.052,-384.627,180.00,-0.00,0.00
C00588=1543.855,0.028,-384.484,-180.00,-0.00,0.00
///RCONF 0,0,0,1,0,0,0,0
C00589=1558.675,8.560,-384.376,180.00,-0.00,0.00
C00590=1570.139,28.367,-384.233,180.00,-0.00,0.00
C00591=1570.159,45.468,-384.126,-180.00,-0.00,0.00
C00592=1558.712,65.341,-383.982,180.00,-0.00,0.00
C00593=1543.913,73.909,-383.875,-180.00,-0.00,0.00
C00594=1520.933,73.932,-383.731,180.00,-0.00,0.00
C00595=1506.113,65.400,-383.624,180.00,-0.00,0.00
C00596=1494.577,45.469,-383.479,180.00,-0.00,0.00
C00597=1494.557,28.367,-383.372,180.00,-0.00,0.00
C00598=1506.841,7.927,-383.223,180.00,-0.00,0.00
///RCONF 0,0,0,0,0,0,0,0
C00599=1520.108,0.247,-383.127,180.00,-0.00,0.00
C00600=1544.767,0.221,-382.972,-180.00,-0.00,0.00
///RCONF 0,0,0,1,0,0,0,0
C00601=1558.051,7.868,-382.876,180.00,-0.00,0.00
C00602=1570.428,29.254,-382.722,180.00,-0.00,0.00
C00603=1570.446,44.579,-382.626,180.00,-0.00,0.00
C00604=1558.090,66.034,-382.471,-180.00,-0.00,0.00
C00605=1544.824,73.714,-382.375,180.00,-0.00,0.00
C00606=1520.021,73.739,-382.220,180.00,-0.00,0.00
C00607=1506.737,66.092,-382.124,180.00,-0.00,0.00
C00608=1494.289,44.582,-381.968,180.00,-0.00,0.00
C00609=1494.270,29.254,-381.872,-180.00,-0.00,0.00
C00610=1507.465,7.234,-381.711,-180.00,-0.00,0.00
///RCONF 0,0,0,0,0,0,0,0
C00611=1519.197,0.442,-381.627,180.00,-0.00,0.00
C00612=1545.679,0.414,-381.461,-180.00,-0.00,0.00
///RCONF 0,0,0,1,0,0,0,0
C00613=1557.428,7.178,-381.376,-180.00,-0.00,0.00
C00614=1570.716,30.140,-381.210,180.00,-0.00,0.00
C00615=1570.733,43.693,-381.126,-180.00,-0.00,0.00
C00616=1557.467,66.727,-380.960,-180.00,-0.00,0.00
C00617=1545.735,73.519,-380.875,-180.00,-0.00,0.00
C00618=1519.109,73.546,-380.708,-180.00,-0.00,0.00
C00619=1507.360,66.782,-380.624,-180.00,-0.00,0.00
C00620=1494.000,43.696,-380.457,180.00,-0.00,0.00
C00621=1493.982,30.143,-380.372,-180.00,-0.00,0.00
C00622=1508.087,6.541,-380.200,-180.00,-0.00,0.00
///RCONF 0,0,0,0,0,0,0,0
C00623=1518.286,0.637,-380.127,-180.00,-0.00,0.00
C00624=1546.591,0.608,-379.950,-180.00,-0.00,0.00
///RCONF 0,0,0,1,0,0,0,0
C00625=1556.800,6.485,-379.876,-180.00,-0.00,0.00
C00626=1571.005,31.027,-379.699,180.00,-0.00,0.00
C00627=1571.019,42.811,-379.626,180.00,-0.00,0.00
C00628=1556.845,67.420,-379.448,-180.00,-0.00,0.00
C00629=1546.646,73.324,-379.375,180.00,-0.00,0.00
C00630=1518.197,73.353,-379.197,180.00,-0.00,0.00
C00631=1507.988,67.475,-379.124,-180.00,-0.00,0.00
C00632=1493.711,42.809,-378.946,-180.00,-0.00,0.00
C00633=1493.697,31.025,-378.872,180.00,-0.00,0.00
C00634=1508.711,5.847,-378.689,180.00,-0.00,0.00
///RCONF 0,0,0,0,0,0,0,0
C00635=1517.374,0.832,-378.627,180.00,-0.00,0.00
C00636=1547.502,0.800,-378.439,180.00,-0.00,0.00
///RCONF 0,0,0,1,0,0,0,0
C00637=1556.177,5.794,-378.376,180.00,-0.00,0.00
C00638=1571.294,31.912,-378.188,180.00,-0.00,0.00
C00639=1571.306,41.919,-378.126,180.00,-0.00,0.00
C00640=1556.220,68.113,-377.937,180.00,-0.00,0.00
C00641=1547.558,73.129,-377.875,180.00,-0.00,0.00
C00642=1517.286,73.161,-377.686,180.00,-0.00,0.00
C00643=1508.611,68.166,-377.624,-180.00,-0.00,0.00
C00644=1493.422,41.924,-377.434,-180.00,-0.00,0.00
C00645=1493.410,31.914,-377.372,180.00,-0.00,0.00
C00646=1509.336,5.154,-377.178,-180.00,-0.00,0.00
///RCONF 0,0,0,0,0,0,0,0
C00647=1516.465,1.026,-377.127,180.00,-0.00,0.00
C00648=1548.414,0.993,-376.928,180.00,-0.00,0.00
///RCONF 0,0,0,1,0,0,0,0
C00649=1555.554,5.103,-376.876,-180.00,-0.00,0.00
C00650=1571.583,32.799,-376.677,-180.00,-0.00,0.00
C00651=1571.593,41.034,-376.626,-180.00,-0.00,0.00
C00652=1555.596,68.807,-376.426,-180.00,-0.00,0.00
C00653=1548.467,72.935,-376.375,-180.00,-0.00,0.00
C00654=1516.373,72.968,-376.175,180.00,-0.00,0.00
C00655=1509.235,68.858,-376.124,180.00,-0.00,0.00
C00656=1493.133,41.037,-375.923,180.00,-0.00,0.00
C00657=1493.122,32.802,-375.872,180.00,-0.00,0.00
C00658=1509.958,4.460,-375.667,180.00,-0.00,0.00
///RCONF 0,0,0,0,0,0,0,0
C00659=1515.554,1.221,-375.627,-180.00,-0.00,0.00
C00660=1549.326,1.186,-375.417,-180.00,-0.00,0.00
///RCONF 0,0,0,1,0,0,0,0
C00661=1554.931,4.413,-375.376,-180.00,-0.00,0.00
C00662=1571.872,33.686,-375.166,180.00,-0.00,0.00
C00663=1571.879,40.152,-375.126,-180.00,-0.00,0.00
C00664=1554.974,69.501,-374.915,-180.00,-0.00,0.00
C00665=1549.378,72.740,-374.875,-180.00,-0.00,0.00
C00666=1515.461,72.774,-374.664,180.00,-0.00,0.00
C00667=1509.857,69.547,-374.624,180.00,-0.00,0.00
C00668=1492.844,40.150,-374.412,180.00,-0.00,0.00
C00669=1492.837,33.684,-374.372,-180.00,-0.00,0.00
C00670=1510.580,3.768,-374.156,-180.00,-0.00,0.00
///RCONF 0,0,0,0,0,0,0,0
C00671=1514.644,1.415,-374.127,-180.00,-0.00,0.00
C00672=1550.237,1.379,-373.906,-180.00,-0.00,0.00
///RCONF 0,0,0,1,0,0,0,0
C00673=1554.306,3.722,-373.876,-180.00,-0.00,0.00
C00674=1572.160,34.570,-373.655,180.00,-0.00,0.00
C00675=1572.166,39.264,-373.626,-180.00,-0.00,0.00
C00676=1554.351,70.193,-373.404,-180.00,-0.00,0.00
C00677=1550.288,72.546,-373.375,-180.00,-0.00,0.00
C00678=1514.550,72.581,-373.153,-180.00,-0.00,0.00
C00679=1510.482,70.238,-373.124,-180.00,-0.00,0.00
C00680=1492.556,39.266,-372.901,-180.00,-0.00,0.00
C00681=1492.550,34.572,-372.872,180.00,-0.00,0.00
C00682=1511.203,3.076,-372.645,180.00,-0.00,0.00
///RCONF 0,0,0,0,0,0,0,0
C00683=1513.732,1.611,-372.627,180.00,-0.00,0.00
C00684=1551.150,1.572,-372.394,-180.00,-0.00,0.00
///RCONF 0,0,0,1,0,0,0,0
C00685=1553.683,3.031,-372.376,180.00,-0.00,0.00
C00686=1572.449,35.457,-372.144,-180.00,-0.00,0.00
C00687=1572.453,38.378,-372.126,180.00,-0.00,0.00
C00688=1553.728,70.887,-371.893,180.00,-0.00,0.00
C00689=1551.200,72.350,-371.875,180.00,-0.00,0.00
C00690=1513.637,72.388,-371.642,180.00,-0.00,0.00
C00691=1511.106,70.931,-371.624,180.00,-0.00,0.00
C00692=1492.267,38.379,-371.390,-180.00,-0.00,0.00
C00693=1492.262,35.460,-371.372,-180.00,-0.00,0.00
///RCONF 0,0,0,0,0,0,0,0
C00694=1511.828,2.381,-371.134,180.00,-0.00,0.00
C00695=1512.821,1.805,-371.127,180.00,-0.00,0.00
C00696=1552.061,1.765,-370.883,180.00,-0.00,0.00
C00697=1553.059,2.339,-370.876,180.00,-0.00,0.00
///RCONF 0,0,0,1,0,0,0,0
C00698=1572.738,36.346,-370.633,180.00,-0.00,0.00
C00699=1572.740,37.490,-370.626,-180.00,-0.00,0.00
C00700=1553.104,71.580,-370.382,180.00,-0.00,0.00
C00701=1552.110,72.155,-370.375,-180.00,-0.00,0.00
C00702=1512.726,72.195,-370.131,-180.00,-0.00,0.00
C00703=1511.731,71.622,-370.124,180.00,-0.00,0.00
C00704=1491.978,37.491,-369.879,180.00,-0.00,0.00
C00705=1491.975,36.346,-369.872,-180.00,-0.00,0.00
///RCONF 0,0,0,0,0,0,0,0
C00706=1512.194,1.868,-369.625,180.00,-0.00,0.00
C00707=1552.676,1.850,-369.375,180.00,-0.00,0.00
///RCONF 0,0,0,1,0,0,0,0
C00708=1572.944,36.918,-369.124,-180.00,-0.00,0.00
C00709=1552.696,72.021,-368.874,180.00,-0.00,0.00
C00710=1512.154,72.039,-368.623,180.00,-0.00,0.00
C00711=1491.855,36.918,-368.372,180.00,-0.00,0.00
C00712=1492.154,36.400,-368.368,180.00,-0.00,0.00
///RCONF 0,0,0,0,0,0,0,0
C00713=1511.847,2.300,-368.124,180.00,-0.00,0.00
C00714=1512.743,1.784,-368.118,-180.00,-0.00,0.00
C00715=1552.117,1.789,-367.874,180.00,-0.00,0.00
C00716=1553.007,2.303,-367.867,180.00,-0.00,0.00
///RCONF 0,0,0,1,0,0,0,0
C00717=1572.692,36.408,-367.623,-180.00,-0.00,0.00
C00718=1572.691,37.428,-367.617,-180.00,-0.00,0.00
C00719=1552.998,71.527,-367.373,-180.00,-0.00,0.00
C00720=1552.117,72.035,-367.366,180.00,-0.00,0.00
C00721=1512.743,72.030,-367.122,180.00,-0.00,0.00
C00722=1511.868,71.524,-367.116,180.00,-0.00,0.00
C00723=1492.183,37.419,-366.872,180.00,-0.00,0.00
C00724=1492.547,35.789,-366.862,-180.00,-0.00,0.00
C00725=1511.514,2.945,-366.625,-180.00,-0.00,0.00
///RCONF 0,0,0,0,0,0,0,0
C00726=1513.468,1.817,-366.611,-180.00,-0.00,0.00
C00727=1551.392,1.823,-366.374,-180.00,-0.00,0.00
///RCONF 0,0,0,1,0,0,0,0
C00728=1553.341,2.949,-366.360,180.00,-0.00,0.00
C00729=1572.300,35.796,-366.124,-180.00,-0.00,0.00
C00730=1572.299,38.039,-366.110,180.00,-0.00,0.00
C00731=1553.331,70.883,-365.873,180.00,-0.00,0.00
C00732=1551.392,72.002,-365.859,180.00,-0.00,0.00
C00733=1513.468,71.996,-365.623,-180.00,-0.00,0.00
C00734=1511.534,70.878,-365.609,-180.00,-0.00,0.00
C00735=1492.575,38.031,-365.372,-180.00,-0.00,0.00
C00736=1492.939,35.175,-365.354,-180.00,-0.00,0.00
C00737=1511.179,3.591,-365.125,-180.00,-0.00,0.00
///RCONF 0,0,0,0,0,0,0,0
C00738=1514.194,1.852,-365.103,180.00,-0.00,0.00
C00739=1550.666,1.857,-364.874,-180.00,-0.00,0.00
///RCONF 0,0,0,1,0,0,0,0
C00740=1553.674,3.595,-364.853,180.00,-0.00,0.00
C00741=1571.908,35.185,-364.624,-180.00,-0.00,0.00
C00742=1571.907,38.653,-364.602,-180.00,-0.00,0.00
C00743=1553.666,70.237,-364.373,180.00,-0.00,0.00
C00744=1550.666,71.967,-364.351,180.00,-0.00,0.00
C00745=1514.194,71.962,-364.123,-180.00,-0.00,0.00
C00746=1511.200,70.232,-364.101,-180.00,-0.00,0.00
C00747=1492.967,38.642,-363.872,180.00,-0.00,0.00
C00748=1493.330,34.564,-363.846,-180.00,-0.00,0.00
C00749=1510.845,4.235,-363.625,-180.00,-0.00,0.00
///RCONF 0,0,0,0,0,0,0,0
C00750=1514.920,1.886,-363.595,-180.00,-0.00,0.00
C00751=1549.941,1.890,-363.374,180.00,-0.00,0.00
///RCONF 0,0,0,1,0,0,0,0
C00752=1554.008,4.240,-363.345,180.00,-0.00,0.00
C00753=1571.516,34.573,-363.124,-180.00,-0.00,0.00
C00754=1571.515,39.264,-363.094,-180.00,-0.00,0.00
C00755=1554.000,69.592,-362.873,180.00,-0.00,0.00
C00756=1549.940,71.934,-362.844,-180.00,-0.00,0.00
C00757=1514.919,71.929,-362.623,180.00,-0.00,0.00
C00758=1510.866,69.587,-362.593,180.00,-0.00,0.00
C00759=1493.359,39.254,-362.372,180.00,-0.00,0.00
C00760=1493.723,33.951,-362.338,-180.00,-0.00,0.00
C00761=1510.511,4.882,-362.125,-180.00,-0.00,0.00
///RCONF 0,0,0,0,0,0,0,0
C00762=1515.646,1.919,-362.088,180.00,-0.00,0.00
C00763=1549.215,1.924,-361.874,180.00,-0.00,0.00
///RCONF 0,0,0,1,0,0,0,0
C00764=1554.343,4.887,-361.837,-180.00,-0.00,0.00
C00765=1571.124,33.960,-361.624,180.00,-0.00,0.00
C00766=1571.122,39.877,-361.586,180.00,-0.00,0.00
C00767=1554.334,68.946,-361.373,180.00,-0.00,0.00
C00768=1549.214,71.900,-361.336,-180.00,-0.00,0.00
C00769=1515.645,71.895,-361.123,-180.00,-0.00,0.00
C00770=1510.531,68.941,-361.085,180.00,-0.00,0.00
C00771=1493.751,39.867,-360.872,180.00,-0.00,0.00
C00772=1494.116,33.339,-360.830,180.00,-0.00,0.00
C00773=1510.178,5.527,-360.625,-180.00,-0.00,0.00
///RCONF 0,0,0,0,0,0,0,0
C00774=1516.373,1.953,-360.580,180.00,-0.00,0.00
C00775=1548.489,1.958,-360.374,180.00,-0.00,0.00
///RCONF 0,0,0,1,0,0,0,0
C00776=1554.678,5.533,-360.329,180.00,-0.00,0.00
C00777=1570.732,33.349,-360.124,-180.00,-0.00,0.00
C00778=1570.729,40.489,-360.078,180.00,-0.00,0.00
C00779=1554.667,68.301,-359.873,-180.00,-0.00,0.00
C00780=1548.487,71.867,-359.828,-180.00,-0.00,0.00
C00781=1516.371,71.861,-359.623,180.00,-0.00,0.00
C00782=1510.197,68.295,-359.577,-180.00,-0.00,0.00
C00783=1494.143,40.478,-359.372,-180.00,-0.00,0.00
C00784=1494.507,32.727,-359.322,-180.00,-0.00,0.00
C00785=1509.844,6.171,-359.125,-180.00,-0.00,0.00
///RCONF 0,0,0,0,0,0,0,0
C00786=1517.099,1.986,-359.071,180.00,-0.00,0.00
C00787=1547.764,1.991,-358.875,-180.00,-0.00,0.00
///RCONF 0,0,0,1,0,0,0,0
C00788=1555.012,6.179,-358.821,-180.00,-0.00,0.00
C00789=1570.340,32.737,-358.624,180.00,-0.00,0.00
C00790=1570.337,41.101,-358.570,180.00,-0.00,0.00
C00791=1555.001,67.656,-358.373,-180.00,-0.00,0.00
C00792=1547.761,71.833,-358.320,180.00,-0.00,0.00
C00793=1517.096,71.828,-358.123,-180.00,-0.00,0.00
C00794=1509.863,67.649,-358.069,-180.00,-0.00,0.00
C00795=1494.535,41.090,-357.872,-180.00,-0.00,0.00
C00796=1494.901,32.115,-357.814,-180.00,-0.00,0.00
C00797=1509.511,6.817,-357.625,180.00,-0.00,0.00
///RCONF 0,0,0,0,0,0,0,0
C00798=1517.821,2.020,-357.563,180.00,-0.00,0.00
C00799=1547.038,2.025,-357.375,180.00,-0.00,0.00
///RCONF 0,0,0,1,0,0,0,0
C00800=1555.344,6.822,-357.313,-180.00,-0.00,0.00
C00801=1569.949,32.127,-357.124,-180.00,-0.00,0.00
C00802=1569.945,41.713,-357.062,180.00,-0.00,0.00
C00803=1555.334,67.011,-356.873,180.00,-0.00,0.00
C00804=1547.039,71.798,-356.811,-180.00,-0.00,0.00
C00805=1517.822,71.794,-356.623,180.00,-0.00,0.00
C00806=1509.530,67.006,-356.561,-180.00,-0.00,0.00
C00807=1494.927,41.702,-356.372,-180.00,-0.00,0.00
C00808=1495.290,31.507,-356.306,180.00,-0.00,0.00
C00809=1509.177,7.462,-356.125,180.00,-0.00,0.00
///RCONF 0,0,0,0,0,0,0,0
C00810=1518.548,2.054,-356.055,180.00,-0.00,0.00
C00811=1546.312,2.058,-355.875,-180.00,-0.00,0.00
///RCONF 0,0,0,1,0,0,0,0
C00812=1555.677,7.466,-355.804,-180.00,-0.00,0.00
C00813=1569.556,31.514,-355.624,180.00,-0.00,0.00
C00814=1569.555,42.321,-355.554,-180.00,-0.00,0.00
C00815=1555.668,66.365,-355.373,-180.00,-0.00,0.00
C00816=1546.312,71.765,-355.303,180.00,-0.00,0.00
C00817=1518.548,71.761,-355.123,180.00,-0.00,0.00
C00818=1509.198,66.361,-355.052,180.00,-0.00,0.00
C00819=1495.319,42.313,-354.872,180.00,-0.00,0.00
C00820=1495.682,30.896,-354.797,-180.00,-0.00,0.00
C00821=1508.843,8.109,-354.625,180.00,-0.00,0.00
///RCONF 0,0,0,0,0,0,0,0
C00822=1519.274,2.088,-354.547,180.00,-0.00,0.00
C00823=1545.586,2.092,-354.375,180.00,-0.00,0.00
///RCONF 0,0,0,1,0,0,0,0
C00824=1556.011,8.113,-354.296,180.00,-0.00,0.00
C00825=1569.164,30.902,-354.124,180.00,-0.00,0.00
C00826=1569.163,42.932,-354.045,180.00,-0.00,0.00
C00827=1556.002,65.719,-353.873,180.00,-0.00,0.00
C00828=1545.586,71.731,-353.795,180.00,-0.00,0.00
C00829=1519.274,71.727,-353.623,-180.00,-0.00,0.00
C00830=1508.863,65.714,-353.544,180.00,-0.00,0.00
C00831=1495.711,42.925,-353.372,-180.00,-0.00,0.00
C00832=1496.075,30.284,-353.289,180.00,-0.00,0.00
C00833=1508.510,8.753,-353.125,-180.00,-0.00,0.00
///RCONF 0,0,0,0,0,0,0,0
C00834=1519.998,2.122,-353.038,-180.00,-0.00,0.00
C00835=1544.861,2.126,-352.875,-180.00,-0.00,0.00
///RCONF 0,0,0,1,0,0,0,0
C00836=1556.345,8.758,-352.787,180.00,-0.00,0.00
C00837=1568.772,30.290,-352.624,-180.00,-0.00,0.00
C00838=1568.770,43.544,-352.537,-180.00,-0.00,0.00
C00839=1556.335,65.075,-352.373,180.00,-0.00,0.00
C00840=1544.862,71.697,-352.286,180.00,-0.00,0.00
C00841=1519.999,71.693,-352.123,-180.00,-0.00,0.00
C00842=1508.529,65.069,-352.035,-180.00,-0.00,0.00
C00843=1496.103,43.537,-351.872,180.00,-0.00,0.00
C00844=1496.467,29.671,-351.780,-180.00,-0.00,0.00
C00845=1508.175,9.399,-351.625,-180.00,-0.00,0.00
///RCONF 0,0,0,0,0,0,0,0
C00846=1520.724,2.156,-351.529,-180.00,-0.00,0.00
C00847=1544.135,2.159,-351.375,180.00,-0.00,0.00
///RCONF 0,0,0,1,0,0,0,0
C00848=1556.678,9.403,-351.279,-180.00,-0.00,0.00
C00849=1568.380,29.679,-351.124,180.00,-0.00,0.00
C00850=1568.378,44.157,-351.028,180.00,-0.00,0.00
C00851=1556.670,64.429,-350.873,-180.00,-0.00,0.00
C00852=1544.136,71.663,-350.777,-180.00,-0.00,0.00
C00853=1520.725,71.660,-350.623,180.00,-0.00,0.00
C00854=1508.196,64.424,-350.527,180.00,-0.00,0.00
C00855=1496.495,44.149,-350.372,180.00,-0.00,0.00
C00856=1496.859,29.061,-350.272,-180.00,-0.00,0.00
C00857=1507.842,10.044,-350.125,-180.00,-0.00,0.00
///RCONF 0,0,0,0,0,0,0,0
C00858=1521.451,2.189,-350.021,-180.00,-0.00,0.00
C00859=1543.409,2.193,-349.875,180.00,-0.00,0.00
///RCONF 0,0,0,1,0,0,0,0
C00860=1557.011,10.049,-349.770,-180.00,-0.00,0.00
C00861=1567.988,29.068,-349.624,-180.00,-0.00,0.00
C00862=1567.986,44.767,-349.519,180.00,-0.00,0.00
C00863=1557.003,63.783,-349.373,180.00,-0.00,0.00
C00864=1543.409,71.629,-349.269,180.00,-0.00,0.00
C00865=1521.451,71.626,-349.123,180.00,-0.00,0.00
C00866=1507.864,63.778,-349.018,-180.00,-0.00,0.00
C00867=1496.887,44.759,-348.872,-180.00,-0.00,0.00
C00868=1497.252,28.450,-348.763,180.00,-0.00,0.00
C00869=1507.509,10.689,-348.625,180.00,-0.00,0.00
///RCONF 0,0,0,0,0,0,0,0
C00870=1522.176,2.224,-348.512,-180.00,-0.00,0.00
C00871=1542.684,2.227,-348.375,-180.00,-0.00,0.00
///RCONF 0,0,0,1,0,0,0,0
C00872=1557.344,10.694,-348.261,180.00,-0.00,0.00
C00873=1567.596,28.455,-348.124,180.00,-0.00,0.00
C00874=1567.594,45.378,-348.011,180.00,-0.00,0.00
C00875=1557.336,63.139,-347.873,180.00,-0.00,0.00
C00876=1542.684,71.595,-347.760,-180.00,-0.00,0.00
C00877=1522.176,71.592,-347.623,-180.00,-0.00,0.00
C00878=1507.530,63.133,-347.509,180.00,-0.00,0.00
C00879=1497.279,45.372,-347.372,180.00,-0.00,0.00
C00880=1497.644,27.838,-347.254,180.00,-0.00,0.00
C00881=1507.174,11.335,-347.125,180.00,-0.00,0.00
///RCONF 0,0,0,0,0,0,0,0
C00882=1522.902,2.258,-347.003,-180.00,-0.00,0.00
C00883=1541.958,2.260,-346.875,180.00,-0.00,0.00
///RCONF 0,0,0,1,0,0,0,0
C00884=1557.679,11.340,-346.752,180.00,-0.00,0.00
C00885=1567.204,27.843,-346.624,-180.00,-0.00,0.00
C00886=1567.202,45.990,-346.502,-180.00,-0.00,0.00
C00887=1557.671,62.493,-346.373,180.00,-0.00,0.00
C00888=1541.958,71.562,-346.251,180.00,-0.00,0.00
C00889=1522.902,71.559,-346.123,-180.00,-0.00,0.00
C00890=1507.195,62.488,-346.000,-180.00,-0.00,0.00
C00891=1497.671,45.984,-345.872,-180.00,-0.00,0.00
C00892=1498.036,27.226,-345.745,-180.00,-0.00,0.00
C00893=1506.840,11.981,-345.625,-180.00,-0.00,0.00
///RCONF 0,0,0,0,0,0,0,0
C00894=1523.628,2.291,-345.494,-180.00,-0.00,0.00
C00895=1541.232,2.294,-345.375,-180.00,-0.00,0.00
///RCONF 0,0,0,1,0,0,0,0
C00896=1558.013,11.986,-345.243,-180.00,-0.00,0.00
C00897=1566.812,27.232,-345.124,180.00,-0.00,0.00
C00898=1566.810,46.602,-344.993,-180.00,-0.00,0.00
C00899=1558.005,61.847,-344.873,-180.00,-0.00,0.00
C00900=1541.232,71.528,-344.742,-180.00,-0.00,0.00
C00901=1523.628,71.525,-344.623,-180.00,-0.00,0.00
C00902=1506.861,61.842,-344.491,180.00,-0.00,0.00
C00903=1498.063,46.595,-344.372,-180.00,-0.00,0.00
C00904=1498.427,26.615,-344.236,180.00,-0.00,0.00
C00905=1506.507,12.624,-344.125,180.00,-0.00,0.00
///RCONF 0,0,0,0,0,0,0,0
C00906=1524.353,2.325,-343.985,-180.00,-0.00,0.00
C00907=1540.506,2.328,-343.875,180.00,-0.00,0.00
///RCONF 0,0,0,1,0,0,0,0
C00908=1558.346,12.630,-343.734,180.00,-0.00,0.00
C00909=1566.420,26.621,-343.624,180.00,-0.00,0.00
C00910=1566.418,47.213,-343.483,180.00,-0.00,0.00
C00911=1558.338,61.203,-343.373,-180.00,-0.00,0.00
C00912=1540.507,71.494,-343.233,-180.00,-0.00,0.00
C00913=1524.354,71.491,-343.123,180.00,-0.00,0.00
C00914=1506.529,61.197,-342.982,180.00,-0.00,0.00
C00915=1498.455,47.206,-342.872,180.00,-0.00,0.00
C00916=1498.820,26.003,-342.726,-180.00,-0.00,0.00
C00917=1506.174,13.270,-342.625,180.00,-0.00,0.00
///RCONF 0,0,0,0,0,0,0,0
C00918=1525.079,2.359,-342.476,180.00,-0.00,0.00
C00919=1539.780,2.361,-342.375,180.00,-0.00,0.00
///RCONF 0,0,0,1,0,0,0,0
C00920=1558.679,13.276,-342.225,-180.00,-0.00,0.00
C00921=1566.028,26.010,-342.124,180.00,-0.00,0.00
C00922=1566.025,47.825,-341.974,180.00,-0.00,0.00
C00923=1558.671,60.558,-341.873,180.00,-0.00,0.00
C00924=1539.781,71.460,-341.724,-180.00,-0.00,0.00
C00925=1525.080,71.458,-341.623,180.00,-0.00,0.00
C00926=1506.195,60.552,-341.473,-180.00,-0.00,0.00
C00927=1498.847,47.819,-341.372,180.00,-0.00,0.00
C00928=1499.212,25.391,-341.217,180.00,-0.00,0.00
C00929=1505.839,13.916,-341.126,180.00,-0.00,0.00
///RCONF 0,0,0,0,0,0,0,0
C00930=1525.805,2.393,-340.966,180.00,-0.00,0.00
C00931=1539.054,2.395,-340.875,-180.00,-0.00,0.00
///RCONF 0,0,0,1,0,0,0,0
C00932=1559.014,13.922,-340.716,180.00,-0.00,0.00
C00933=1565.636,25.397,-340.624,-180.00,-0.00,0.00
C00934=1565.633,48.437,-340.465,-180.00,-0.00,0.00
C00935=1559.006,59.911,-340.373,-180.00,-0.00,0.00
C00936=1539.055,71.426,-340.214,180.00,-0.00,0.00
C00937=1525.806,71.424,-340.123,-180.00,-0.00,0.00
C00938=1505.861,59.906,-339.964,-180.00,-0.00,0.00
C00939=1499.239,48.430,-339.872,-180.00,-0.00,0.00
C00940=1499.605,24.779,-339.708,-180.00,-0.00,0.00
C00941=1505.505,14.562,-339.626,180.00,-0.00,0.00
///RCONF 0,0,0,0,0,0,0,0
C00942=1526.530,2.427,-339.457,180.00,-0.00,0.00
C00943=1538.330,2.429,-339.375,180.00,-0.00,0.00
///RCONF 0,0,0,1,0,0,0,0
C00944=1559.347,14.566,-339.206,-180.00,-0.00,0.00
C00945=1565.244,24.785,-339.124,180.00,-0.00,0.00
C00946=1565.241,49.049,-338.955,-180.00,-0.00,0.00
C00947=1559.339,59.266,-338.873,-180.00,-0.00,0.00
C00948=1538.330,71.392,-338.705,180.00,-0.00,0.00
C00949=1526.530,71.390,-338.623,-180.00,-0.00,0.00
C00950=1505.528,59.261,-338.454,-180.00,-0.00,0.00
C00951=1499.631,49.042,-338.372,-180.00,-0.00,0.00
C00952=1499.996,24.168,-338.198,-180.00,-0.00,0.00
C00953=1505.172,15.205,-338.126,180.00,-0.00,0.00
///RCONF 0,0,0,0,0,0,0,0
C00954=1527.256,2.461,-337.947,180.00,-0.00,0.00
C00955=1537.603,2.462,-337.875,180.00,-0.00,0.00
///RCONF 0,0,0,1,0,0,0,0
C00956=1559.680,15.212,-337.696,-180.00,-0.00,0.00
C00957=1564.852,24.173,-337.624,-180.00,-0.00,0.00
C00958=1564.849,49.660,-337.446,180.00,-0.00,0.00
C00959=1559.673,58.622,-337.373,180.00,-0.00,0.00
C00960=1537.604,71.359,-337.195,-180.00,-0.00,0.00
C00961=1527.257,71.357,-337.123,180.00,-0.00,0.00
C00962=1505.194,58.615,-336.944,-180.00,-0.00,0.00
C00963=1500.023,49.654,-336.872,180.00,-0.00,0.00
C00964=1500.389,23.556,-336.688,-180.00,-0.00,0.00
C00965=1504.838,15.853,-336.626,-180.00,-0.00,0.00
C00966=1527.982,2.494,-336.437,180.00,-0.00,0.00
C00967=1536.877,2.496,-336.375,-180.00,-0.00,0.00
C00968=1560.014,15.858,-336.187,180.00,-0.00,0.00
C00969=1564.460,23.562,-336.124,-180.00,-0.00,0.00
C00970=1564.457,50.271,-335.936,180.00,-0.00,0.00
C00971=1560.007,57.976,-335.873,180.00,-0.00,0.00
C00972=1536.878,71.325,-335.685,180.00,-0.00,0.00
C00973=1527.983,71.323,-335.623,180.00,-0.00,0.00
C00974=1504.860,57.969,-335.435,-180.00,-0.00,0.00
C00975=1500.415,50.265,-335.372,-180.00,-0.00,0.00
C00976=1500.781,22.945,-335.178,180.00,-0.00,0.00
C00977=1504.504,16.497,-335.126,-180.00,-0.00,0.00
C00978=1528.708,2.529,-334.928,180.00,-0.00,0.00
C00979=1536.152,2.530,-334.875,180.00,-0.00,0.00
C00980=1560.347,16.503,-334.677,180.00,-0.00,0.00
C00981=1564.068,22.950,-334.624,-180.00,-0.00,0.00
C00982=1564.064,50.883,-334.426,-180.00,-0.00,0.00
C00983=1560.341,57.330,-334.373,180.00,-0.00,0.00
C00984=1536.152,71.290,-334.175,180.00,-0.00,0.00
C00985=1528.708,71.289,-334.123,180.00,-0.00,0.00
C00986=1504.527,57.324,-333.925,180.00,-0.00,0.00
C00987=1500.807,50.877,-333.872,180.00,-0.00,0.00
C00988=1501.173,22.333,-333.668,-180.00,-0.00,0.00
C00989=1504.171,17.142,-333.626,180.00,-0.00,0.00
C00990=1529.433,2.562,-333.418,-180.00,-0.00,0.00
C00991=1535.427,2.563,-333.375,-180.00,-0.00,0.00
C00992=1560.680,17.147,-333.167,-180.00,-0.00,0.00
C00993=1563.676,22.338,-333.124,180.00,-0.00,0.00
C00994=1563.672,51.495,-332.916,-180.00,-0.00,0.00
C00995=1560.674,56.686,-332.873,-180.00,-0.00,0.00
C00996=1535.427,71.257,-332.665,-180.00,-0.00,0.00
C00997=1529.433,71.256,-332.623,180.00,-0.00,0.00
C00998=1504.194,56.680,-332.415,-180.00,-0.00,0.00
C00999=1501.199,51.489,-332.372,-180.00,-0.00,0.00
C01000=1501.566,21.721,-332.158,-180.00,-0.00,0.00
C01001=1503.836,17.788,-332.126,-180.00,-0.00,0.00
C01002=1530.159,2.596,-331.907,-180.00,-0.00,0.00
C01003=1534.701,2.597,-331.875,180.00,-0.00,0.00
C01004=1561.015,17.794,-331.657,-180.00,-0.00,0.00
C01005=1563.284,21.727,-331.624,-180.00,-0.00,0.00
C01006=1563.280,52.107,-331.406,180.00,-0.00,0.00
C01007=1561.009,56.039,-331.373,-180.00,-0.00,0.00
C01008=1534.701,71.223,-331.155,180.00,-0.00,0.00
C01009=1530.159,71.222,-331.123,-180.00,-0.00,0.00
C01010=1503.860,56.034,-330.905,180.00,-0.00,0.00
C01011=1501.591,52.101,-330.872,-180.00,-0.00,0.00
C01012=1501.957,21.110,-330.648,-180.00,-0.00,0.00
C01013=1503.503,18.433,-330.626,-180.00,-0.00,0.00
C01014=1530.885,2.630,-330.397,-180.00,-0.00,0.00
C01015=1533.975,2.631,-330.375,180.00,-0.00,0.00
C01016=1561.347,18.439,-330.146,-180.00,-0.00,0.00
C01017=1562.892,21.115,-330.124,180.00,-0.00,0.00
C01018=1562.888,52.717,-329.896,180.00,-0.00,0.00
C01019=1561.342,55.395,-329.873,-180.00,-0.00,0.00
C01020=1533.975,71.189,-329.645,-180.00,-0.00,0.00
C01021=1530.885,71.188,-329.623,180.00,-0.00,0.00
C01022=1503.527,55.389,-329.394,-180.00,-0.00,0.00
C01023=1501.983,52.712,-329.372,180.00,-0.00,0.00
C01024=1502.350,20.498,-329.138,180.00,-0.00,0.00
C01025=1503.170,19.078,-329.126,-180.00,-0.00,0.00
C01026=1531.611,2.664,-328.887,180.00,-0.00,0.00
C01027=1533.249,2.664,-328.875,180.00,-0.00,0.00
C01028=1561.681,19.084,-328.636,180.00,-0.00,0.00
C01029=1562.500,20.503,-328.624,-180.00,-0.00,0.00
C01030=1562.495,53.330,-328.385,-180.00,-0.00,0.00
C01031=1561.675,54.750,-328.373,-180.00,-0.00,0.00
C01032=1533.249,71.155,-328.135,-180.00,-0.00,0.00
C01033=1531.611,71.155,-328.123,-180.00,-0.00,0.00
C01034=1503.193,54.744,-327.884,180.00,-0.00,0.00
C01035=1502.375,53.324,-327.872,-180.00,-0.00,0.00
C01036=1502.741,19.887,-327.627,-180.00,-0.00,0.00
C01037=1502.835,19.724,-327.626,-180.00,-0.00,0.00
C01038=1532.336,2.698,-327.376,180.00,-0.00,0.00
C01039=1532.523,2.698,-327.375,-180.00,-0.00,0.00
C01040=1562.014,19.729,-327.125,180.00,-0.00,0.00
C01041=1562.108,19.891,-327.124,-180.00,-0.00,0.00
C01042=1562.104,53.941,-326.875,-180.00,-0.00,0.00
C01043=1562.010,54.102,-326.873,180.00,-0.00,0.00
C01044=1532.523,71.121,-326.624,180.00,-0.00,0.00
C01045=1532.337,71.121,-326.623,180.00,-0.00,0.00
C01046=1502.860,54.098,-326.373,-180.00,-0.00,0.00
C01047=1502.768,53.935,-326.372,-180.00,-0.00,0.00
C01048=1502.812,20.125,-326.124,180.00,-0.00,0.00
C01049=1503.076,19.665,-326.120,-180.00,-0.00,0.00
C01050=1532.184,2.910,-325.873,-180.00,-0.00,0.00
C01051=1532.671,2.909,-325.870,180.00,-0.00,0.00
C01052=1561.739,19.742,-325.623,180.00,-0.00,0.00
C01053=1561.959,20.125,-325.620,180.00,-0.00,0.00
C01054=1561.915,53.711,-325.373,180.00,-0.00,0.00
C01055=1561.716,54.054,-325.370,-180.00,-0.00,0.00
C01056=1532.609,70.810,-325.124,-180.00,-0.00,0.00
C01057=1532.255,70.811,-325.121,180.00,-0.00,0.00
C01058=1503.187,53.979,-324.874,180.00,-0.00,0.00
C01059=1503.034,53.710,-324.872,180.00,-0.00,0.00
C01060=1503.066,20.893,-324.629,180.00,-0.00,0.00
C01061=1503.872,19.503,-324.617,180.00,-0.00,0.00
C01062=1531.642,3.505,-324.379,180.00,-0.00,0.00
C01063=1533.217,3.507,-324.367,-180.00,-0.00,0.00
C01064=1560.957,19.558,-324.129,180.00,-0.00,0.00
C01065=1561.727,20.894,-324.118,180.00,-0.00,0.00
C01066=1561.694,52.943,-323.880,-180.00,-0.00,0.00
C01067=1560.938,54.248,-323.869,-180.00,-0.00,0.00
C01068=1533.168,70.246,-323.631,-180.00,-0.00,0.00
C01069=1531.692,70.243,-323.620,-180.00,-0.00,0.00
C01070=1503.953,54.192,-323.383,180.00,-0.00,0.00
C01071=1503.233,52.942,-323.372,-180.00,-0.00,0.00
C01072=1503.264,21.663,-323.137,180.00,-0.00,0.00
C01073=1504.634,19.291,-323.117,-180.00,-0.00,0.00
C01074=1531.073,4.061,-322.888,180.00,-0.00,0.00
C01075=1533.783,4.062,-322.867,-180.00,-0.00,0.00
C01076=1560.193,19.346,-322.638,180.00,-0.00,0.00
C01077=1561.528,21.662,-322.618,-180.00,-0.00,0.00
C01078=1561.496,52.173,-322.389,180.00,-0.00,0.00
C01079=1560.176,54.460,-322.369,180.00,-0.00,0.00
C01080=1533.737,69.689,-322.140,-180.00,-0.00,0.00
C01081=1531.126,69.688,-322.120,-180.00,-0.00,0.00
C01082=1504.716,54.405,-321.891,-180.00,-0.00,0.00
C01083=1503.432,52.174,-321.872,-180.00,-0.00,0.00
C01084=1503.461,22.435,-321.646,180.00,-0.00,0.00
C01085=1505.400,19.079,-321.617,180.00,-0.00,0.00
C01086=1530.508,4.615,-321.396,-180.00,-0.00,0.00
C01087=1534.350,4.619,-321.367,180.00,-0.00,0.00
C01088=1559.429,19.132,-321.147,180.00,-0.00,0.00
C01089=1561.329,22.431,-321.118,180.00,-0.00,0.00
C01090=1561.300,51.401,-320.898,180.00,-0.00,0.00
C01091=1559.410,54.672,-320.869,-180.00,-0.00,0.00
C01092=1534.302,69.135,-320.649,-180.00,-0.00,0.00
C01093=1530.559,69.131,-320.620,180.00,-0.00,0.00
C01094=1505.481,54.618,-320.400,180.00,-0.00,0.00
C01095=1503.631,51.405,-320.372,180.00,-0.00,0.00
C01096=1503.659,23.201,-320.155,-180.00,-0.00,0.00
C01097=1506.167,18.865,-320.116,-180.00,-0.00,0.00
C01098=1529.939,5.172,-319.905,-180.00,-0.00,0.00
C01099=1534.916,5.175,-319.867,180.00,-0.00,0.00
C01100=1558.664,18.919,-319.656,180.00,-0.00,0.00
C01101=1561.130,23.199,-319.618,-180.00,-0.00,0.00
C01102=1561.102,50.635,-319.407,-180.00,-0.00,0.00
C01103=1558.643,54.886,-319.369,180.00,-0.00,0.00
C01104=1534.872,68.578,-319.158,-180.00,-0.00,0.00
C01105=1529.993,68.575,-319.120,180.00,-0.00,0.00
C01106=1506.245,54.832,-318.909,180.00,-0.00,0.00
C01107=1503.830,50.636,-318.872,180.00,-0.00,0.00
C01108=1503.857,23.974,-318.664,180.00,-0.00,0.00
C01109=1506.929,18.654,-318.616,-180.00,-0.00,0.00
C01110=1529.375,5.726,-318.415,-180.00,-0.00,0.00
C01111=1535.483,5.732,-318.367,180.00,-0.00,0.00
C01112=1557.899,18.705,-318.165,180.00,-0.00,0.00
C01113=1560.931,23.968,-318.118,180.00,-0.00,0.00
C01114=1560.904,49.862,-317.916,180.00,-0.00,0.00
C01115=1557.881,55.097,-317.869,-180.00,-0.00,0.00
C01116=1535.435,68.024,-317.667,-180.00,-0.00,0.00
C01117=1529.426,68.018,-317.620,180.00,-0.00,0.00
C01118=1507.010,55.045,-317.419,180.00,-0.00,0.00
C01119=1504.029,49.867,-317.372,-180.00,-0.00,0.00
C01120=1504.055,24.739,-317.174,180.00,-0.00,0.00
C01121=1507.698,18.440,-317.116,180.00,-0.00,0.00
C01122=1528.806,6.283,-316.924,-180.00,-0.00,0.00
C01123=1536.050,6.289,-316.867,-180.00,-0.00,0.00
C01124=1557.133,18.490,-316.675,-180.00,-0.00,0.00
C01125=1560.732,24.737,-316.618,180.00,-0.00,0.00
C01126=1560.707,49.097,-316.426,180.00,-0.00,0.00
C01127=1557.112,55.311,-316.369,-180.00,-0.00,0.00
C01128=1536.004,67.468,-316.177,-180.00,-0.00,0.00
C01129=1528.859,67.461,-316.120,-180.00,-0.00,0.00
C01130=1507.776,55.260,-315.928,180.00,-0.00,0.00
C01131=1504.227,49.098,-315.872,-180.00,-0.00,0.00
C01132=1504.251,25.508,-315.683,-180.00,-0.00,0.00
C01133=1508.463,18.228,-315.616,-180.00,-0.00,0.00
C01134=1528.240,6.837,-315.434,180.00,-0.00,0.00
C01135=1536.616,6.845,-315.367,-180.00,-0.00,0.00
C01136=1556.368,18.277,-315.184,-180.00,-0.00,0.00
C01137=1560.534,25.507,-315.118,-180.00,-0.00,0.00
C01138=1560.510,48.328,-314.935,180.00,-0.00,0.00
C01139=1556.348,55.523,-314.869,-180.00,-0.00,0.00
C01140=1536.571,66.913,-314.686,-180.00,-0.00,0.00
C01141=1528.293,66.905,-314.620,-180.00,-0.00,0.00
C01142=1508.541,55.473,-314.438,180.00,-0.00,0.00
C01143=1504.426,48.328,-314.372,-180.00,-0.00,0.00
C01144=1504.449,26.277,-314.193,180.00,-0.00,0.00
C01145=1509.229,18.016,-314.116,-180.00,-0.00,0.00
C01146=1527.673,7.393,-313.944,-180.00,-0.00,0.00
C01147=1537.183,7.402,-313.867,180.00,-0.00,0.00
C01148=1555.602,18.062,-313.694,180.00,-0.00,0.00
C01149=1560.335,26.275,-313.618,180.00,-0.00,0.00
C01150=1560.312,47.559,-313.445,180.00,-0.00,0.00
C01151=1555.582,55.735,-313.369,-180.00,-0.00,0.00
C01152=1537.137,66.358,-313.196,180.00,-0.00,0.00
C01153=1527.726,66.348,-313.120,180.00,-0.00,0.00
C01154=1509.307,55.688,-312.948,-180.00,-0.00,0.00
C01155=1504.625,47.560,-312.872,-180.00,-0.00,0.00
C01156=1504.647,27.046,-312.704,180.00,-0.00,0.00
C01157=1509.994,17.804,-312.616,-180.00,-0.00,0.00
C01158=1527.102,7.950,-312.454,180.00,-0.00,0.00
C01159=1537.749,7.958,-312.367,180.00,-0.00,0.00
C01160=1554.840,17.850,-312.205,-180.00,-0.00,0.00
C01161=1560.136,27.044,-312.118,180.00,-0.00,0.00
C01162=1560.115,46.790,-311.956,180.00,-0.00,0.00
C01163=1554.817,55.947,-311.869,180.00,-0.00,0.00
C01164=1537.708,65.801,-311.707,180.00,-0.00,0.00
C01165=1527.160,65.792,-311.620,180.00,-0.00,0.00
C01166=1510.069,55.899,-311.458,180.00,-0.00,0.00
C01167=1504.824,46.791,-311.372,-180.00,-0.00,0.00
C01168=1504.844,27.814,-311.214,-180.00,-0.00,0.00
C01169=1510.759,17.591,-311.116,-180.00,-0.00,0.00
C01170=1526.538,8.503,-310.965,180.00,-0.00,0.00
C01171=1538.316,8.515,-310.867,180.00,-0.00,0.00
C01172=1554.075,17.637,-310.715,-180.00,-0.00,0.00
C01173=1559.938,27.817,-310.618,-180.00,-0.00,0.00
C01174=1559.917,46.022,-310.466,180.00,-0.00,0.00
C01175=1554.052,56.160,-310.369,-180.00,-0.00,0.00
C01176=1538.273,65.247,-310.217,180.00,-0.00,0.00
C01177=1526.593,65.235,-310.120,-180.00,-0.00,0.00
C01178=1510.834,56.114,-309.969,180.00,-0.00,0.00
C01179=1505.021,46.018,-309.872,180.00,-0.00,0.00
C01180=1505.040,28.586,-309.725,180.00,-0.00,0.00
C01181=1511.523,17.380,-309.616,180.00,-0.00,0.00
C01182=1525.968,9.060,-309.475,-180.00,-0.00,0.00
C01183=1538.882,9.071,-309.367,180.00,-0.00,0.00
C01184=1553.311,17.423,-309.226,180.00,-0.00,0.00
C01185=1559.739,28.582,-309.118,-180.00,-0.00,0.00
C01186=1559.721,45.250,-308.977,180.00,-0.00,0.00
C01187=1553.288,56.371,-308.869,-180.00,-0.00,0.00
C01188=1538.842,64.690,-308.728,-180.00,-0.00,0.00
C01189=1526.027,64.679,-308.620,-180.00,-0.00,0.00
C01190=1511.598,56.327,-308.480,-180.00,-0.00,0.00
C01191=1505.221,45.254,-308.372,-180.00,-0.00,0.00
C01192=1505.238,29.355,-308.236,-180.00,-0.00,0.00
C01193=1512.290,17.166,-308.116,180.00,-0.00,0.00
C01194=1525.403,9.614,-307.987,-180.00,-0.00,0.00
C01195=1539.449,9.628,-307.866,-180.00,-0.00,0.00
C01196=1552.546,17.209,-307.737,-180.00,-0.00,0.00
C01197=1559.540,29.350,-307.617,-180.00,-0.00,0.00
C01198=1559.523,44.481,-307.488,-180.00,-0.00,0.00
C01199=1552.521,56.585,-307.369,180.00,-0.00,0.00
C01200=1539.407,64.137,-307.239,-180.00,-0.00,0.00
C01201=1525.460,64.122,-307.120,-180.00,-0.00,0.00
C01202=1512.364,56.541,-306.991,180.00,-0.00,0.00
C01203=1505.420,44.485,-306.872,-180.00,-0.00,0.00
C01204=1505.436,30.125,-306.748,180.00,-0.00,0.00
C01205=1513.053,16.955,-306.616,180.00,-0.00,0.00
C01206=1524.833,10.170,-306.498,180.00,-0.00,0.00
C01207=1540.015,10.184,-306.366,180.00,-0.00,0.00
C01208=1551.782,16.996,-306.249,-180.00,-0.00,0.00
C01209=1559.341,30.119,-306.117,180.00,-0.00,0.00
C01210=1559.325,43.711,-306.000,180.00,-0.00,0.00
C01211=1551.758,56.796,-305.869,-180.00,-0.00,0.00
C01212=1539.977,63.580,-305.751,-180.00,-0.00,0.00
C01213=1524.894,63.566,-305.620,180.00,-0.00,0.00
C01214=1513.127,56.754,-305.502,180.00,-0.00,0.00
C01215=1505.619,43.716,-305.372,-180.00,-0.00,0.00
C01216=1505.633,30.889,-305.259,180.00,-0.00,0.00
C01217=1513.819,16.742,-305.116,-180.00,-0.00,0.00
C01218=1524.269,10.725,-305.010,180.00,-0.00,0.00
C01219=1540.582,10.741,-304.866,-180.00,-0.00,0.00
C01220=1551.017,16.782,-304.760,180.00,-0.00,0.00
C01221=1559.142,30.888,-304.617,180.00,-0.00,0.00
C01222=1559.128,42.947,-304.511,-180.00,-0.00,0.00
C01223=1550.991,57.009,-304.369,-180.00,-0.00,0.00
C01224=1540.542,63.026,-304.263,-180.00,-0.00,0.00
C01225=1524.327,63.009,-304.120,-180.00,-0.00,0.00
C01226=1513.892,56.969,-304.014,180.00,-0.00,0.00
C01227=1505.818,42.947,-303.872,180.00,-0.00,0.00
C01228=1505.831,31.662,-303.771,-180.00,-0.00,0.00
C01229=1514.586,16.528,-303.616,180.00,-0.00,0.00
C01230=1523.701,11.280,-303.522,180.00,-0.00,0.00
C01231=1541.149,11.298,-303.366,180.00,-0.00,0.00
C01232=1550.252,16.568,-303.272,-180.00,-0.00,0.00
C01233=1558.943,31.655,-303.117,180.00,-0.00,0.00
C01234=1558.931,42.174,-303.023,-180.00,-0.00,0.00
C01235=1550.225,57.222,-302.869,180.00,-0.00,0.00
C01236=1541.109,62.471,-302.775,-180.00,-0.00,0.00
C01237=1523.760,62.452,-302.620,180.00,-0.00,0.00
C01238=1514.657,57.182,-302.526,180.00,-0.00,0.00
C01239=1506.016,42.180,-302.372,-180.00,-0.00,0.00
C01240=1506.027,32.428,-302.284,-180.00,-0.00,0.00
C01241=1515.351,16.317,-302.115,180.00,-0.00,0.00
C01242=1523.135,11.834,-302.034,-180.00,-0.00,0.00
C01243=1541.714,11.854,-301.866,-180.00,-0.00,0.00
C01244=1549.488,16.354,-301.785,180.00,-0.00,0.00
C01245=1558.745,32.424,-301.617,180.00,-0.00,0.00
C01246=1558.734,41.408,-301.536,-180.00,-0.00,0.00
C01247=1549.460,57.434,-301.368,-180.00,-0.00,0.00
C01248=1541.675,61.916,-301.287,-180.00,-0.00,0.00
C01249=1523.195,61.896,-301.120,180.00,-0.00,0.00
C01250=1515.421,57.395,-301.039,-180.00,-0.00,0.00
C01251=1506.215,41.411,-300.872,180.00,-0.00,0.00
C01252=1506.224,33.197,-300.797,-180.00,-0.00,0.00
C01253=1516.116,16.105,-300.615,180.00,-0.00,0.00
C01254=1522.566,12.390,-300.547,180.00,-0.00,0.00
C01255=1542.282,12.411,-300.366,180.00,-0.00,0.00
C01256=1548.724,16.141,-300.298,-180.00,-0.00,0.00
C01257=1558.546,33.195,-300.117,-180.00,-0.00,0.00
C01258=1558.537,40.639,-300.049,180.00,-0.00,0.00
C01259=1548.694,57.647,-299.868,180.00,-0.00,0.00
C01260=1542.244,61.360,-299.800,-180.00,-0.00,0.00
C01261=1522.627,61.339,-299.620,180.00,-0.00,0.00
C01262=1516.186,57.609,-299.552,180.00,-0.00,0.00
C01263=1506.412,40.637,-299.372,-180.00,-0.00,0.00
C01264=1506.420,33.965,-299.310,180.00,-0.00,0.00
C01265=1516.880,15.892,-299.115,-180.00,-0.00,0.00
C01266=1521.999,12.945,-299.060,180.00,-0.00,0.00
C01267=1542.848,12.967,-298.866,180.00,-0.00,0.00
C01268=1547.961,15.928,-298.811,180.00,-0.00,0.00
C01269=1558.347,33.964,-298.617,-180.00,-0.00,0.00
C01270=1558.340,39.871,-298.562,-180.00,-0.00,0.00
C01271=1547.931,57.859,-298.368,180.00,-0.00,0.00
C01272=1542.811,60.806,-298.313,180.00,-0.00,0.00
C01273=1522.061,60.783,-298.120,-180.00,-0.00,0.00
C01274=1516.949,57.823,-298.065,180.00,-0.00,0.00
C01275=1506.611,39.870,-297.872,180.00,-0.00,0.00
C01276=1506.617,34.733,-297.823,180.00,-0.00,0.00
C01277=1517.647,15.679,-297.615,180.00,-0.00,0.00
C01278=1521.432,13.500,-297.574,-180.00,-0.00,0.00
C01279=1543.414,13.524,-297.366,-180.00,-0.00,0.00
C01280=1547.194,15.713,-297.325,180.00,-0.00,0.00
C01281=1558.148,34.732,-297.117,180.00,-0.00,0.00
C01282=1558.143,39.101,-297.076,180.00,-0.00,0.00
C01283=1547.164,58.071,-296.868,-180.00,-0.00,0.00
C01284=1543.378,60.251,-296.827,180.00,-0.00,0.00
C01285=1521.495,60.226,-296.620,180.00,-0.00,0.00
C01286=1517.715,58.037,-296.579,-180.00,-0.00,0.00
C01287=1506.810,39.102,-296.372,180.00,-0.00,0.00
C01288=1506.814,35.502,-296.337,-180.00,-0.00,0.00
C01289=1518.412,15.468,-296.115,180.00,-0.00,0.00
C01290=1520.864,14.055,-296.088,180.00,-0.00,0.00
C01291=1543.980,14.080,-295.866,180.00,-0.00,0.00
C01292=1546.431,15.501,-295.839,-180.00,-0.00,0.00
C01293=1557.950,35.501,-295.617,-180.00,-0.00,0.00
C01294=1557.946,38.333,-295.590,180.00,-0.00,0.00
C01295=1546.398,58.284,-295.368,180.00,-0.00,0.00
C01296=1543.946,59.695,-295.341,-180.00,-0.00,0.00
C01297=1520.929,59.670,-295.120,180.00,-0.00,0.00
C01298=1518.478,58.250,-295.093,180.00,-0.00,0.00
C01299=1507.008,38.330,-294.872,180.00,-0.00,0.00
C01300=1507.010,36.273,-294.852,180.00,-0.00,0.00
C01301=1519.176,15.255,-294.615,180.00,-0.00,0.00
C01302=1520.297,14.610,-294.602,-180.00,-0.00,0.00
C01303=1544.548,14.637,-294.366,-180.00,-0.00,0.00
C01304=1545.666,15.285,-294.353,-180.00,-0.00,0.00
C01305=1557.750,36.271,-294.117,180.00,-0.00,0.00
C01306=1557.749,37.562,-294.104,-180.00,-0.00,0.00
C01307=1545.635,58.496,-293.868,-180.00,-0.00,0.00
C01308=1544.513,59.140,-293.856,180.00,-0.00,0.00
C01309=1520.361,59.113,-293.620,180.00,-0.00,0.00
C01310=1519.243,58.465,-293.607,180.00,-0.00,0.00
C01311=1507.209,37.565,-293.372,180.00,-0.00,0.00
C01312=1519.843,15.114,-293.116,180.00,-0.00,0.00
C01313=1544.995,15.153,-292.867,180.00,-0.00,0.00
C01314=1557.516,36.917,-292.617,-180.00,-0.00,0.00
C01315=1544.950,58.606,-292.368,-180.00,-0.00,0.00
C01316=1519.931,58.567,-292.120,-180.00,-0.00,0.00
C01317=1507.479,36.918,-291.872,180.00,-0.00,0.00
C01318=1519.699,15.805,-291.626,-180.00,-0.00,0.00
C01319=1519.878,15.571,-291.623,180.00,-0.00,0.00
C01320=1520.177,15.372,-291.620,180.00,-0.00,0.00
C01321=1520.487,15.335,-291.616,180.00,-0.00,0.00
C01322=1544.373,15.362,-291.376,180.00,-0.00,0.00
C01323=1544.912,15.556,-291.370,-180.00,-0.00,0.00
C01324=1544.925,15.602,-291.370,-180.00,-0.00,0.00
C01325=1545.137,15.817,-291.367,-180.00,-0.00,0.00
C01326=1557.087,36.570,-291.125,-180.00,-0.00,0.00
C01327=1557.089,37.263,-291.118,-180.00,-0.00,0.00
C01328=1545.092,57.991,-290.877,-180.00,-0.00,0.00
C01329=1544.813,58.168,-290.874,180.00,-0.00,0.00
C01330=1544.683,58.274,-290.872,-180.00,-0.00,0.00
C01331=1544.373,58.419,-290.869,-180.00,-0.00,0.00
C01332=1520.487,58.393,-290.628,180.00,-0.00,0.00
C01333=1520.104,58.190,-290.623,-180.00,-0.00,0.00
C01334=1520.104,58.136,-290.623,180.00,-0.00,0.00
C01335=1519.792,57.978,-290.619,180.00,-0.00,0.00
C01336=1507.843,37.225,-290.378,180.00,-0.00,0.00
C01337=1507.842,36.614,-290.372,-180.00,-0.00,0.00
C01338=1519.484,16.486,-290.135,-180.00,-0.00,0.00
C01339=1519.663,16.251,-290.132,180.00,-0.00,0.00
C01340=1519.702,16.162,-290.131,-180.00,-0.00,0.00
C01341=1520.811,15.521,-290.118,180.00,-0.00,0.00
C01342=1520.890,15.531,-290.117,180.00,-0.00,0.00
C01343=1521.190,15.494,-290.114,-180.00,-0.00,0.00
C01344=1543.670,15.514,-289.886,180.00,-0.00,0.00
C01345=1543.970,15.586,-289.882,180.00,-0.00,0.00
C01346=1544.047,15.568,-289.882,-180.00,-0.00,0.00
C01347=1545.113,16.187,-289.869,180.00,-0.00,0.00
C01348=1545.142,16.282,-289.868,-180.00,-0.00,0.00
C01349=1545.355,16.496,-289.865,-180.00,-0.00,0.00
C01350=1556.612,36.037,-289.635,180.00,-0.00,0.00
C01351=1556.612,37.797,-289.618,180.00,-0.00,0.00
C01352=1545.319,57.319,-289.388,-180.00,-0.00,0.00
C01353=1545.042,57.496,-289.385,-180.00,-0.00,0.00
C01354=1545.031,57.601,-289.384,-180.00,-0.00,0.00
C01355=1544.049,58.168,-289.372,180.00,-0.00,0.00
C01356=1543.970,58.131,-289.371,180.00,-0.00,0.00
C01357=1543.670,58.278,-289.368,180.00,-0.00,0.00
C01358=1521.190,58.258,-289.139,-180.00,-0.00,0.00
C01359=1520.890,58.076,-289.135,-180.00,-0.00,0.00
C01360=1520.813,58.120,-289.135,180.00,-0.00,0.00
C01361=1519.873,57.576,-289.123,180.00,-0.00,0.00
C01362=1519.872,57.465,-289.122,180.00,-0.00,0.00
C01363=1519.561,57.307,-289.119,180.00,-0.00,0.00
C01364=1508.303,37.766,-288.889,180.00,-0.00,0.00
C01365=1508.305,36.071,-288.872,-180.00,-0.00,0.00
C01366=1519.248,17.152,-288.647,-180.00,-0.00,0.00
C01367=1519.425,16.916,-288.644,180.00,-0.00,0.00
C01368=1519.465,16.828,-288.643,-180.00,-0.00,0.00
C01369=1521.484,15.654,-288.618,-180.00,-0.00,0.00
C01370=1521.537,15.661,-288.618,180.00,-0.00,0.00
C01371=1521.868,15.624,-288.615,-180.00,-0.00,0.00
C01372=1542.992,15.642,-288.397,180.00,-0.00,0.00
C01373=1543.323,15.714,-288.393,-180.00,-0.00,0.00
C01374=1543.376,15.701,-288.393,180.00,-0.00,0.00
C01375=1545.349,16.854,-288.369,180.00,-0.00,0.00
C01376=1545.377,16.948,-288.368,180.00,-0.00,0.00
C01377=1545.590,17.163,-288.365,180.00,-0.00,0.00
C01378=1556.152,35.497,-288.147,-180.00,-0.00,0.00
C01379=1556.150,38.337,-288.117,180.00,-0.00,0.00
C01380=1545.556,56.652,-287.899,180.00,-0.00,0.00
C01381=1545.279,56.830,-287.896,-180.00,-0.00,0.00
C01382=1545.268,56.935,-287.895,180.00,-0.00,0.00
C01383=1543.376,58.028,-287.872,180.00,-0.00,0.00
C01384=1543.323,58.001,-287.872,180.00,-0.00,0.00
C01385=1542.992,58.148,-287.868,-180.00,-0.00,0.00
C01386=1521.868,58.129,-287.650,-180.00,-0.00,0.00
C01387=1521.537,57.948,-287.646,180.00,-0.00,0.00
C01388=1521.484,57.981,-287.646,180.00,-0.00,0.00
C01389=1519.638,56.909,-287.624,-180.00,-0.00,0.00
C01390=1519.638,56.798,-287.622,180.00,-0.00,0.00
C01391=1519.325,56.640,-287.619,180.00,-0.00,0.00
C01392=1508.763,38.307,-287.401,-180.00,-0.00,0.00
C01393=1508.766,35.531,-287.372,-180.00,-0.00,0.00
C01394=1519.006,17.829,-287.158,-180.00,-0.00,0.00
C01395=1519.169,17.612,-287.156,-180.00,-0.00,0.00
C01396=1519.214,17.513,-287.154,180.00,-0.00,0.00
C01397=1522.201,15.781,-287.118,-180.00,-0.00,0.00
C01398=1522.282,15.791,-287.117,180.00,-0.00,0.00
C01399=1522.587,15.753,-287.114,180.00,-0.00,0.00
C01400=1542.273,15.770,-286.909,180.00,-0.00,0.00
C01401=1542.578,15.842,-286.905,180.00,-0.00,0.00
C01402=1542.658,15.824,-286.904,180.00,-0.00,0.00
C01403=1545.599,17.539,-286.869,180.00,-0.00,0.00
C01404=1545.633,17.645,-286.868,-180.00,-0.00,0.00
C01405=1545.832,17.840,-286.865,180.00,-0.00,0.00
C01406=1555.692,34.956,-286.658,180.00,-0.00,0.00
C01407=1555.689,38.877,-286.618,-180.00,-0.00,0.00
C01408=1545.798,55.976,-286.411,-180.00,-0.00,0.00
C01409=1545.540,56.137,-286.408,180.00,-0.00,0.00
C01410=1545.524,56.253,-286.407,180.00,-0.00,0.00
C01411=1542.659,57.906,-286.372,180.00,-0.00,0.00
C01412=1542.578,57.868,-286.371,-180.00,-0.00,0.00
C01413=1542.273,58.019,-286.368,180.00,-0.00,0.00
C01414=1522.587,58.001,-286.162,-180.00,-0.00,0.00
C01415=1522.282,57.817,-286.158,180.00,-0.00,0.00
C01416=1522.202,57.863,-286.157,180.00,-0.00,0.00
C01417=1519.383,56.226,-286.123,-180.00,-0.00,0.00
C01418=1519.379,56.104,-286.122,180.00,-0.00,0.00
C01419=1519.084,55.963,-286.119,180.00,-0.00,0.00
C01420=1509.224,38.847,-285.912,180.00,-0.00,0.00
C01421=1509.227,34.991,-285.872,-180.00,-0.00,0.00
C01422=1518.779,18.479,-285.670,-180.00,-0.00,0.00
C01423=1518.956,18.236,-285.667,180.00,-0.00,0.00
C01424=1518.990,18.160,-285.666,180.00,-0.00,0.00
C01425=1522.891,15.911,-285.618,180.00,-0.00,0.00
C01426=1522.955,15.919,-285.618,-180.00,-0.00,0.00
C01427=1523.271,15.882,-285.614,180.00,-0.00,0.00
C01428=1541.589,15.898,-285.420,180.00,-0.00,0.00
C01429=1541.905,15.966,-285.417,180.00,-0.00,0.00
C01430=1541.969,15.952,-285.416,180.00,-0.00,0.00
C01431=1545.819,18.188,-285.369,180.00,-0.00,0.00
C01432=1545.843,18.270,-285.368,180.00,-0.00,0.00
C01433=1546.058,18.491,-285.365,-180.00,-0.00,0.00
C01434=1555.232,34.416,-285.170,-180.00,-0.00,0.00
C01435=1555.228,39.417,-285.117,180.00,-0.00,0.00
C01436=1546.026,55.325,-284.923,180.00,-0.00,0.00
C01437=1545.751,55.512,-284.919,-180.00,-0.00,0.00
C01438=1545.742,55.602,-284.918,-180.00,-0.00,0.00
C01439=1541.969,57.774,-284.872,-180.00,-0.00,0.00
C01440=1541.905,57.742,-284.871,180.00,-0.00,0.00
C01441=1541.589,57.890,-284.868,-180.00,-0.00,0.00
C01442=1523.271,57.873,-284.674,180.00,-0.00,0.00
C01443=1522.955,57.694,-284.670,180.00,-0.00,0.00
C01444=1522.891,57.733,-284.669,-180.00,-0.00,0.00
C01445=1519.168,55.574,-284.624,-180.00,-0.00,0.00
C01446=1519.170,55.477,-284.623,180.00,-0.00,0.00
C01447=1518.857,55.312,-284.619,180.00,-0.00,0.00
C01448=1509.684,39.388,-284.424,-180.00,-0.00,0.00
C01449=1509.688,34.451,-284.372,-180.00,-0.00,0.00
C01450=1518.542,19.145,-284.182,-180.00,-0.00,0.00
C01451=1518.719,18.898,-284.179,180.00,-0.00,0.00
C01452=1518.753,18.824,-284.178,-180.00,-0.00,0.00
C01453=1523.596,16.039,-284.118,-180.00,-0.00,0.00
C01454=1523.666,16.048,-284.117,-180.00,-0.00,0.00
C01455=1523.973,16.011,-284.114,-180.00,-0.00,0.00
C01456=1540.887,16.026,-283.933,-180.00,-0.00,0.00
C01457=1541.194,16.093,-283.929,180.00,-0.00,0.00
C01458=1541.264,16.078,-283.928,180.00,-0.00,0.00
C01459=1546.053,18.854,-283.869,180.00,-0.00,0.00
C01460=1546.077,18.934,-283.868,180.00,-0.00,0.00
C01461=1546.294,19.157,-283.865,-180.00,-0.00,0.00
C01462=1554.772,33.875,-283.683,-180.00,-0.00,0.00
C01463=1554.767,39.957,-283.617,180.00,-0.00,0.00
C01464=1546.263,54.660,-283.435,180.00,-0.00,0.00
C01465=1545.987,54.849,-283.431,180.00,-0.00,0.00
C01466=1545.977,54.937,-283.430,-180.00,-0.00,0.00
C01467=1541.264,57.647,-283.372,180.00,-0.00,0.00
C01468=1541.194,57.612,-283.371,180.00,-0.00,0.00
C01469=1540.887,57.761,-283.368,-180.00,-0.00,0.00
C01470=1523.973,57.746,-283.186,180.00,-0.00,0.00
C01471=1523.666,57.568,-283.182,180.00,-0.00,0.00
C01472=1523.596,57.609,-283.181,-180.00,-0.00,0.00
C01473=1518.936,54.907,-283.124,180.00,-0.00,0.00
C01474=1518.938,54.813,-283.123,180.00,-0.00,0.00
C01475=1518.621,54.646,-283.119,-180.00,-0.00,0.00
C01476=1510.144,39.928,-282.937,-180.00,-0.00,0.00
C01477=1510.149,33.911,-282.872,-180.00,-0.00,0.00
C01478=1518.298,19.823,-282.695,-180.00,-0.00,0.00
C01479=1518.457,19.601,-282.692,-180.00,-0.00,0.00
C01480=1518.499,19.514,-282.691,180.00,-0.00,0.00
C01481=1524.300,16.168,-282.618,180.00,-0.00,0.00
C01482=1524.367,16.176,-282.617,180.00,-0.00,0.00
C01483=1524.665,16.140,-282.614,180.00,-0.00,0.00
C01484=1540.195,16.154,-282.445,-180.00,-0.00,0.00
C01485=1540.493,16.217,-282.442,-180.00,-0.00,0.00
C01486=1540.560,16.203,-282.441,-180.00,-0.00,0.00
C01487=1546.308,19.543,-282.369,180.00,-0.00,0.00
C01488=1546.338,19.637,-282.368,-180.00,-0.00,0.00
C01489=1546.537,19.836,-282.365,-180.00,-0.00,0.00
C01490=1554.311,33.335,-282.195,180.00,-0.00,0.00
C01491=1554.306,40.497,-282.117,180.00,-0.00,0.00
C01492=1546.506,53.981,-281.948,-180.00,-0.00,0.00
C01493=1546.253,54.149,-281.944,-180.00,-0.00,0.00
C01494=1546.238,54.252,-281.943,-180.00,-0.00,0.00
C01495=1540.560,57.521,-281.872,180.00,-0.00,0.00
C01496=1540.493,57.489,-281.871,180.00,-0.00,0.00
C01497=1540.195,57.632,-281.868,180.00,-0.00,0.00
C01498=1524.665,57.617,-281.699,180.00,-0.00,0.00
C01499=1524.367,57.448,-281.695,-180.00,-0.00,0.00
C01500=1524.300,57.485,-281.694,-180.00,-0.00,0.00
C01501=1518.675,54.222,-281.623,180.00,-0.00,0.00
C01502=1518.672,54.112,-281.622,-180.00,-0.00,0.00
C01503=1518.379,53.967,-281.619,-180.00,-0.00,0.00
C01504=1510.604,40.469,-281.449,180.00,-0.00,0.00
C01505=1510.610,33.371,-281.372,180.00,-0.00,0.00
C01506=1518.062,20.490,-281.208,-180.00,-0.00,0.00
C01507=1518.219,20.266,-281.205,-180.00,-0.00,0.00
C01508=1518.262,20.180,-281.204,180.00,-0.00,0.00
C01509=1525.007,16.297,-281.118,-180.00,-0.00,0.00
C01510=1525.083,16.306,-281.117,-180.00,-0.00,0.00
C01511=1525.370,16.270,-281.114,-180.00,-0.00,0.00
C01512=1539.490,16.283,-280.958,180.00,-0.00,0.00
C01513=1539.777,16.343,-280.955,-180.00,-0.00,0.00
C01514=1539.852,16.329,-280.954,180.00,-0.00,0.00
C01515=1546.543,20.211,-280.869,-180.00,-0.00,0.00
C01516=1546.572,20.304,-280.868,180.00,-0.00,0.00
C01517=1546.772,20.503,-280.865,180.00,-0.00,0.00
C01518=1553.851,32.793,-280.708,-180.00,-0.00,0.00
C01519=1553.845,41.038,-280.617,180.00,-0.00,0.00
C01520=1546.743,53.315,-280.461,180.00,-0.00,0.00
C01521=1546.490,53.483,-280.457,180.00,-0.00,0.00
C01522=1546.475,53.585,-280.456,-180.00,-0.00,0.00
C01523=1539.853,57.395,-280.372,180.00,-0.00,0.00
C01524=1539.777,57.359,-280.371,180.00,-0.00,0.00
C01525=1539.490,57.502,-280.368,180.00,-0.00,0.00
C01526=1525.370,57.489,-280.212,-180.00,-0.00,0.00
C01527=1525.083,57.322,-280.208,-180.00,-0.00,0.00
C01528=1525.008,57.362,-280.207,180.00,-0.00,0.00
C01529=1518.440,53.554,-280.123,-180.00,-0.00,0.00
C01530=1518.438,53.445,-280.122,-180.00,-0.00,0.00
C01531=1518.143,53.300,-280.119,180.00,-0.00,0.00
C01532=1511.064,41.010,-279.962,-180.00,-0.00,0.00
C01533=1511.071,32.830,-279.872,180.00,-0.00,0.00
C01534=1517.823,21.159,-279.721,180.00,-0.00,0.00
C01535=1517.980,20.934,-279.718,180.00,-0.00,0.00
C01536=1518.023,20.845,-279.717,180.00,-0.00,0.00
C01537=1525.694,16.427,-279.618,180.00,-0.00,0.00
C01538=1525.747,16.433,-279.617,-180.00,-0.00,0.00
C01539=1526.048,16.399,-279.614,180.00,-0.00,0.00
C01540=1538.812,16.411,-279.471,180.00,-0.00,0.00
C01541=1539.113,16.467,-279.468,180.00,-0.00,0.00
C01542=1539.166,16.457,-279.467,180.00,-0.00,0.00
C01543=1546.779,20.878,-279.369,180.00,-0.00,0.00
C01544=1546.809,20.974,-279.368,-180.00,-0.00,0.00
C01545=1547.010,21.173,-279.364,-180.00,-0.00,0.00
C01546=1553.391,32.253,-279.221,180.00,-0.00,0.00
C01547=1553.384,41.578,-279.117,180.00,-0.00,0.00
C01548=1546.981,52.645,-278.974,-180.00,-0.00,0.00
C01549=1546.728,52.815,-278.971,-180.00,-0.00,0.00
C01550=1546.713,52.919,-278.969,180.00,-0.00,0.00
C01551=1539.166,57.260,-278.872,180.00,-0.00,0.00
C01552=1539.113,57.235,-278.871,180.00,-0.00,0.00
C01553=1538.812,57.373,-278.868,180.00,-0.00,0.00
C01554=1526.048,57.361,-278.725,180.00,-0.00,0.00
C01555=1525.747,57.201,-278.721,-180.00,-0.00,0.00
C01556=1525.694,57.230,-278.720,180.00,-0.00,0.00
C01557=1518.204,52.887,-278.624,180.00,-0.00,0.00
C01558=1518.203,52.775,-278.622,-180.00,-0.00,0.00
C01559=1517.906,52.630,-278.619,-180.00,-0.00,0.00
C01560=1511.524,41.551,-278.476,180.00,-0.00,0.00
C01561=1511.532,32.290,-278.372,180.00,-0.00,0.00
C01562=1517.594,21.812,-278.235,180.00,-0.00,0.00
C01563=1517.753,21.579,-278.231,180.00,-0.00,0.00
C01564=1517.786,21.510,-278.231,-180.00,-0.00,0.00
C01565=1526.401,16.555,-278.118,180.00,-0.00,0.00
C01566=1526.466,16.563,-278.117,-180.00,-0.00,0.00
C01567=1526.755,16.528,-278.114,180.00,-0.00,0.00
C01568=1538.105,16.539,-277.985,-180.00,-0.00,0.00
C01569=1538.394,16.594,-277.982,180.00,-0.00,0.00
C01570=1538.458,16.582,-277.981,-180.00,-0.00,0.00
C01571=1547.013,21.544,-277.869,180.00,-0.00,0.00
C01572=1547.035,21.619,-277.868,-180.00,-0.00,0.00
C01573=1547.238,21.827,-277.864,180.00,-0.00,0.00
C01574=1552.931,31.712,-277.735,180.00,-0.00,0.00
C01575=1552.923,42.118,-277.617,180.00,-0.00,0.00
C01576=1547.211,51.992,-277.488,-180.00,-0.00,0.00
C01577=1546.960,52.172,-277.484,180.00,-0.00,0.00
C01578=1546.948,52.254,-277.483,180.00,-0.00,0.00
C01579=1538.459,57.135,-277.372,180.00,-0.00,0.00
C01580=1538.394,57.105,-277.371,-180.00,-0.00,0.00
C01581=1538.105,57.244,-277.367,-180.00,-0.00,0.00
C01582=1526.755,57.233,-277.239,180.00,-0.00,0.00
C01583=1526.466,57.074,-277.235,180.00,-0.00,0.00
C01584=1526.402,57.108,-277.234,-180.00,-0.00,0.00
C01585=1517.972,52.220,-277.124,180.00,-0.00,0.00
C01586=1517.972,52.131,-277.123,-180.00,-0.00,0.00
C01587=1517.677,51.976,-277.119,-180.00,-0.00,0.00
C01588=1511.984,42.092,-276.989,-180.00,-0.00,0.00
C01589=1511.993,31.750,-276.872,-180.00,-0.00,0.00
C01590=1517.357,22.478,-276.749,180.00,-0.00,0.00
C01591=1517.517,22.238,-276.745,-180.00,-0.00,0.00
C01592=1517.549,22.173,-276.745,180.00,-0.00,0.00
C01593=1527.112,16.683,-276.618,-180.00,-0.00,0.00
C01594=1527.169,16.689,-276.617,-180.00,-0.00,0.00
C01595=1527.444,16.657,-276.614,-180.00,-0.00,0.00
C01596=1537.416,16.667,-276.499,180.00,-0.00,0.00
C01597=1537.691,16.716,-276.496,180.00,-0.00,0.00
C01598=1537.747,16.706,-276.495,-180.00,-0.00,0.00
C01599=1547.246,22.208,-276.369,180.00,-0.00,0.00
C01600=1547.267,22.281,-276.368,-180.00,-0.00,0.00
C01601=1547.474,22.493,-276.364,180.00,-0.00,0.00
C01602=1552.471,31.171,-276.249,-180.00,-0.00,0.00
C01603=1552.462,42.658,-276.117,180.00,-0.00,0.00
C01604=1547.447,51.326,-276.002,180.00,-0.00,0.00
C01605=1547.194,51.512,-275.998,-180.00,-0.00,0.00
C01606=1547.183,51.590,-275.997,-180.00,-0.00,0.00
C01607=1537.748,57.011,-275.872,-180.00,-0.00,0.00
C01608=1537.691,56.986,-275.871,180.00,-0.00,0.00
C01609=1537.416,57.115,-275.868,180.00,-0.00,0.00
C01610=1527.444,57.105,-275.753,-180.00,-0.00,0.00
C01611=1527.169,56.959,-275.749,-180.00,-0.00,0.00
C01612=1527.113,56.987,-275.748,-180.00,-0.00,0.00
C01613=1517.741,51.554,-275.624,180.00,-0.00,0.00
C01614=1517.741,51.469,-275.623,180.00,-0.00,0.00
C01615=1517.442,51.310,-275.619,180.00,-0.00,0.00
C01616=1512.444,42.632,-275.503,180.00,-0.00,0.00
C01617=1512.454,31.210,-275.372,-180.00,-0.00,0.00
C01618=1517.120,23.146,-275.263,180.00,-0.00,0.00
C01619=1517.279,22.904,-275.260,-180.00,-0.00,0.00
C01620=1517.313,22.837,-275.259,180.00,-0.00,0.00
C01621=1527.825,16.811,-275.117,-180.00,-0.00,0.00
C01622=1527.934,16.823,-275.116,-180.00,-0.00,0.00
C01623=1528.185,16.787,-275.113,-180.00,-0.00,0.00
C01624=1536.675,16.795,-275.014,-180.00,-0.00,0.00
C01625=1536.926,16.847,-275.011,180.00,-0.00,0.00
C01626=1537.033,16.832,-275.010,-180.00,-0.00,0.00
C01627=1547.480,22.874,-274.869,180.00,-0.00,0.00
C01628=1547.501,22.948,-274.868,-180.00,-0.00,0.00
C01629=1547.710,23.162,-274.864,-180.00,-0.00,0.00
C01630=1552.012,30.631,-274.764,180.00,-0.00,0.00
C01631=1552.001,43.198,-274.617,-180.00,-0.00,0.00
C01632=1547.685,50.658,-274.516,-180.00,-0.00,0.00
C01633=1547.430,50.846,-274.513,-180.00,-0.00,0.00
C01634=1547.419,50.926,-274.512,180.00,-0.00,0.00
C01635=1537.035,56.888,-274.372,-180.00,-0.00,0.00
C01636=1536.926,56.842,-274.370,180.00,-0.00,0.00
C01637=1536.675,56.985,-274.367,180.00,-0.00,0.00
C01638=1528.185,56.977,-274.268,-180.00,-0.00,0.00
C01639=1527.934,56.818,-274.264,180.00,-0.00,0.00
C01640=1527.827,56.867,-274.263,180.00,-0.00,0.00
C01641=1517.507,50.888,-274.124,180.00,-0.00,0.00
C01642=1517.509,50.801,-274.123,-180.00,-0.00,0.00
C01643=1517.205,50.641,-274.119,-180.00,-0.00,0.00
C01644=1512.904,43.173,-274.018,180.00,-0.00,0.00
C01645=1512.915,30.670,-273.872,-180.00,-0.00,0.00
C01646=1516.869,23.837,-273.778,180.00,-0.00,0.00
C01647=1516.996,23.643,-273.776,180.00,-0.00,0.00
C01648=1517.045,23.549,-273.774,-180.00,-0.00,0.00
C01649=1528.510,16.942,-273.617,-180.00,-0.00,0.00
C01650=1528.585,16.950,-273.617,180.00,-0.00,0.00
C01651=1528.855,16.916,-273.613,-180.00,-0.00,0.00
C01652=1536.005,16.923,-273.529,180.00,-0.00,0.00
C01653=1536.275,16.971,-273.525,-180.00,-0.00,0.00
C01654=1536.349,16.960,-273.524,180.00,-0.00,0.00
C01655=1547.751,23.583,-273.368,180.00,-0.00,0.00
C01656=1547.786,23.687,-273.367,180.00,-0.00,0.00
C01657=1547.960,23.853,-273.364,180.00,-0.00,0.00
C01658=1551.552,30.090,-273.279,180.00,-0.00,0.00
C01659=1551.540,43.738,-273.117,180.00,-0.00,0.00
C01660=1547.936,49.968,-273.031,-180.00,-0.00,0.00
C01661=1547.723,50.112,-273.028,180.00,-0.00,0.00
C01662=1547.700,50.221,-273.027,180.00,-0.00,0.00
C01663=1536.350,56.753,-272.872,180.00,-0.00,0.00
C01664=1536.275,56.719,-272.871,-180.00,-0.00,0.00
C01665=1536.005,56.856,-272.867,180.00,-0.00,0.00
C01666=1528.855,56.849,-272.783,-180.00,-0.00,0.00
C01667=1528.585,56.698,-272.779,-180.00,-0.00,0.00
C01668=1528.511,56.735,-272.778,180.00,-0.00,0.00
C01669=1517.223,50.186,-272.623,180.00,-0.00,0.00
C01670=1517.214,50.068,-272.622,-180.00,-0.00,0.00
C01671=1516.955,49.950,-272.618,180.00,-0.00,0.00
C01672=1513.364,43.713,-272.533,-180.00,-0.00,0.00
C01673=1513.376,30.130,-272.372,180.00,-0.00,0.00
C01674=1516.679,24.420,-272.292,-180.00,-0.00,0.00
C01675=1529.477,17.045,-272.114,-180.00,-0.00,0.00
C01676=1535.382,17.051,-272.043,180.00,-0.00,0.00
C01677=1548.145,24.433,-271.865,180.00,-0.00,0.00
C01678=1551.092,29.551,-271.794,180.00,-0.00,0.00
C01679=1551.079,44.278,-271.617,-180.00,-0.00,0.00
C01680=1548.125,49.384,-271.546,180.00,-0.00,0.00
C01681=1535.383,56.727,-271.368,-180.00,-0.00,0.00
C01682=1529.478,56.721,-271.297,180.00,-0.00,0.00
C01683=1516.771,49.370,-271.120,180.00,-0.00,0.00
C01684=1513.823,44.253,-271.049,180.00,-0.00,0.00
C01685=1513.837,29.590,-270.872,-180.00,-0.00,0.00
C01686=1516.441,25.088,-270.808,-180.00,-0.00,0.00
C01687=1530.175,17.174,-270.614,-180.00,-0.00,0.00
C01688=1534.682,17.178,-270.559,180.00,-0.00,0.00
C01689=1548.382,25.103,-270.365,-180.00,-0.00,0.00
C01690=1550.633,29.011,-270.310,180.00,-0.00,0.00
C01691=1550.618,44.818,-270.117,-180.00,-0.00,0.00
C01692=1548.363,48.716,-270.061,180.00,-0.00,0.00
C01693=1534.685,56.598,-269.868,-180.00,-0.00,0.00
C01694=1530.178,56.593,-269.813,180.00,-0.00,0.00
C01695=1516.533,48.700,-269.620,-180.00,-0.00,0.00
C01696=1514.283,44.793,-269.565,180.00,-0.00,0.00
C01697=1514.298,29.050,-269.372,-180.00,-0.00,0.00
C01698=1516.203,25.757,-269.325,180.00,-0.00,0.00
C01699=1530.875,17.303,-269.114,-180.00,-0.00,0.00
C01700=1533.984,17.306,-269.075,180.00,-0.00,0.00
C01701=1548.619,25.772,-268.865,-180.00,-0.00,0.00
C01702=1550.172,28.469,-268.826,180.00,-0.00,0.00
C01703=1550.157,45.359,-268.616,-180.00,-0.00,0.00
C01704=1548.601,48.048,-268.578,-180.00,-0.00,0.00
C01705=1533.985,56.469,-268.368,-180.00,-0.00,0.00
C01706=1530.876,56.465,-268.329,180.00,-0.00,0.00
C01707=1516.296,48.031,-268.120,180.00,-0.00,0.00
C01708=1514.743,45.335,-268.081,180.00,-0.00,0.00
C01709=1514.759,28.509,-267.872,180.00,-0.00,0.00
C01710=1515.966,26.423,-267.842,-180.00,-0.00,0.00
C01711=1531.572,17.433,-267.614,-180.00,-0.00,0.00
C01712=1533.286,17.435,-267.592,-180.00,-0.00,0.00
C01713=1548.858,26.443,-267.365,180.00,-0.00,0.00
C01714=1549.712,27.927,-267.343,-180.00,-0.00,0.00
C01715=1549.697,45.898,-267.116,-180.00,-0.00,0.00
C01716=1548.838,47.381,-267.095,180.00,-0.00,0.00
C01717=1533.288,56.339,-266.868,-180.00,-0.00,0.00
C01718=1531.574,56.337,-266.846,180.00,-0.00,0.00
C01719=1516.058,47.360,-266.620,180.00,-0.00,0.00
C01720=1515.203,45.876,-266.598,-180.00,-0.00,0.00
C01721=1515.220,27.970,-266.372,180.00,-0.00,0.00
C01722=1515.728,27.091,-266.365,180.00,-0.00,0.00
C01723=1532.271,17.562,-266.231,180.00,-0.00,0.00
C01724=1532.589,17.562,-266.228,180.00,-0.00,0.00
C01725=1549.095,27.112,-266.094,180.00,-0.00,0.00
C01726=1549.253,27.388,-266.092,180.00,-0.00,0.00
C01727=1549.236,46.437,-265.958,-180.00,-0.00,0.00
C01728=1549.076,46.713,-265.956,180.00,-0.00,0.00
C01729=1532.589,56.210,-265.822,-180.00,-0.00,0.00
C01730=1532.271,56.209,-265.820,-180.00,-0.00,0.00
C01731=1515.820,46.691,-265.686,-180.00,-0.00,0.00
C01732=1515.662,46.416,-265.684,-180.00,-0.00,0.00
C01733=1515.681,27.431,-265.550,180.00,-0.00,0.00
C01734=1515.840,27.155,-265.550,-180.00,-0.00,0.00
C01735=1532.271,17.669,-265.550,-180.00,-0.00,0.00
C01736=1532.589,17.670,-265.550,180.00,-0.00,0.00
C01737=1549.021,27.156,-265.550,-180.00,-0.00,0.00
C01738=1549.179,27.431,-265.550,180.00,-0.00,0.00
C01739=1549.179,46.405,-265.550,180.00,-0.00,0.00
C01740=1549.020,46.681,-265.550,180.00,-0.00,0.00
C01741=1532.589,56.167,-265.550,-180.00,-0.00,0.00
C01742=1532.271,56.166,-265.550,180.00,-0.00,0.00
C01743=1515.839,46.680,-265.550,180.00,-0.00,0.00
C01744=1515.839,46.680,-165.550,180.00,-0.00,0.00
//INST
///DATE 2023/03/01 09:55
///COMM Generated using RoboDK
///ATTR SC,RW
///GROUP1 RB1
NOP
'Program generated by RoboDK v
'5.5.4 for GP88 Robot on 01/03
'/2023 09:55:42
'Using nominal kinematics.
'Using FRAME-MESA (targets wrt
' base):
'1032.4,-463.1,-432.9,0.0,0.0,
'0.0
'Tool extrusora_teste should b
'e close to:
'-2.5,412.5,61.7,0.0,-90.0,-90
'.0
'Show extrusora_teste
MOVJ C00000 VJ=50.00 PL=0
MOVL C00001 V=150.0 PL=0
MOVL C00002 V=20.0 PL=0
MOVL C00003 V=20.0 PL=0
MOVL C00004 V=20.0 PL=0
MOVL C00005 V=20.0 PL=0
MOVL C00006 V=20.0 PL=0
MOVL C00007 V=20.0 PL=0
MOVL C00008 V=20.0 PL=0
MOVL C00009 V=20.0 PL=0
MOVL C00010 V=20.0 PL=0
MOVL C00011 V=20.0 PL=0
MOVL C00012 V=20.0 PL=0
MOVL C00013 V=20.0 PL=0
MOVL C00014 V=20.0 PL=0
MOVL C00015 V=20.0 PL=0
MOVL C00016 V=20.0 PL=0
MOVL C00017 V=20.0 PL=0
MOVL C00018 V=20.0 PL=0
MOVL C00019 V=20.0 PL=0
MOVL C00020 V=20.0 PL=0
MOVL C00021 V=20.0 PL=0
MOVL C00022 V=20.0 PL=0
MOVL C00023 V=20.0 PL=0
MOVL C00024 V=20.0 PL=0
MOVL C00025 V=20.0 PL=0
MOVL C00026 V=20.0 PL=0
MOVL C00027 V=20.0 PL=0
MOVL C00028 V=20.0 PL=0
MOVL C00029 V=20.0 PL=0
MOVL C00030 V=20.0 PL=0
MOVL C00031 V=20.0 PL=0
MOVL C00032 V=20.0 PL=0
MOVL C00033 V=20.0 PL=0
MOVL C00034 V=20.0 PL=0
MOVL C00035 V=20.0 PL=0
MOVL C00036 V=20.0 PL=0
MOVL C00037 V=20.0 PL=0
MOVL C00038 V=20.0 PL=0
MOVL C00039 V=20.0 PL=0
MOVL C00040 V=20.0 PL=0
MOVL C00041 V=20.0 PL=0
MOVL C00042 V=20.0 PL=0
MOVL C00043 V=20.0 PL=0
MOVL C00044 V=20.0 PL=0
MOVL C00045 V=20.0 PL=0
MOVL C00046 V=20.0 PL=0
MOVL C00047 V=20.0 PL=0
MOVL C00048 V=20.0 PL=0
MOVL C00049 V=20.0 PL=0
MOVL C00050 V=20.0 PL=0
MOVL C00051 V=20.0 PL=0
MOVL C00052 V=20.0 PL=0
MOVL C00053 V=20.0 PL=0
MOVL C00054 V=20.0 PL=0
MOVL C00055 V=20.0 PL=0
MOVL C00056 V=20.0 PL=0
MOVL C00057 V=20.0 PL=0
MOVL C00058 V=20.0 PL=0
MOVL C00059 V=20.0 PL=0
MOVL C00060 V=20.0 PL=0
MOVL C00061 V=20.0 PL=0
MOVL C00062 V=20.0 PL=0
MOVL C00063 V=20.0 PL=0
MOVL C00064 V=20.0 PL=0
MOVL C00065 V=20.0 PL=0
MOVL C00066 V=20.0 PL=0
MOVL C00067 V=20.0 PL=0
MOVL C00068 V=20.0 PL=0
MOVL C00069 V=20.0 PL=0
MOVL C00070 V=20.0 PL=0
MOVL C00071 V=150.0 PL=0
MOVL C00072 V=20.0 PL=0
MOVL C00073 V=20.0 PL=0
MOVL C00074 V=20.0 PL=0
MOVL C00075 V=20.0 PL=0
MOVL C00076 V=20.0 PL=0
MOVL C00077 V=20.0 PL=0
MOVL C00078 V=20.0 PL=0
MOVL C00079 V=20.0 PL=0
MOVL C00080 V=20.0 PL=0
MOVL C00081 V=20.0 PL=0
MOVL C00082 V=20.0 PL=0
MOVL C00083 V=20.0 PL=0
MOVL C00084 V=20.0 PL=0
MOVL C00085 V=150.0 PL=0
MOVL C00086 V=150.0 PL=0
MOVL C00087 V=150.0 PL=0
MOVL C00088 V=20.0 PL=0
MOVL C00089 V=20.0 PL=0
MOVL C00090 V=20.0 PL=0
MOVL C00091 V=20.0 PL=0
MOVL C00092 V=20.0 PL=0
MOVL C00093 V=20.0 PL=0
MOVL C00094 V=150.0 PL=0
MOVL C00095 V=20.0 PL=0
MOVL C00096 V=20.0 PL=0
MOVL C00097 V=150.0 PL=0
MOVL C00098 V=20.0 PL=0
MOVL C00099 V=150.0 PL=0
MOVL C00100 V=20.0 PL=0
MOVL C00101 V=20.0 PL=0
MOVL C00102 V=150.0 PL=0
MOVL C00103 V=20.0 PL=0
MOVL C00104 V=150.0 PL=0
MOVL C00105 V=20.0 PL=0
MOVL C00106 V=20.0 PL=0
MOVL C00107 V=150.0 PL=0
MOVL C00108 V=20.0 PL=0
MOVL C00109 V=150.0 PL=0
MOVL C00110 V=20.0 PL=0
MOVL C00111 V=150.0 PL=0
MOVL C00112 V=20.0 PL=0
MOVL C00113 V=150.0 PL=0
MOVL C00114 V=20.0 PL=0
MOVL C00115 V=150.0 PL=0
MOVL C00116 V=20.0 PL=0
MOVL C00117 V=150.0 PL=0
MOVL C00118 V=20.0 PL=0
MOVL C00119 V=150.0 PL=0
MOVL C00120 V=20.0 PL=0
MOVL C00121 V=150.0 PL=0
MOVL C00122 V=20.0 PL=0
MOVL C00123 V=150.0 PL=0
MOVL C00124 V=20.0 PL=0
MOVL C00125 V=150.0 PL=0
MOVL C00126 V=20.0 PL=0
MOVL C00127 V=150.0 PL=0
MOVL C00128 V=20.0 PL=0
MOVL C00129 V=150.0 PL=0
MOVL C00130 V=20.0 PL=0
MOVL C00131 V=150.0 PL=0
MOVL C00132 V=20.0 PL=0
MOVL C00133 V=150.0 PL=0
MOVL C00134 V=20.0 PL=0
MOVL C00135 V=150.0 PL=0
MOVL C00136 V=20.0 PL=0
MOVL C00137 V=150.0 PL=0
MOVL C00138 V=20.0 PL=0
MOVL C00139 V=150.0 PL=0
MOVL C00140 V=20.0 PL=0
MOVL C00141 V=150.0 PL=0
MOVL C00142 V=20.0 PL=0
MOVL C00143 V=150.0 PL=0
MOVL C00144 V=20.0 PL=0
MOVL C00145 V=150.0 PL=0
MOVL C00146 V=20.0 PL=0
MOVL C00147 V=150.0 PL=0
MOVL C00148 V=20.0 PL=0
MOVL C00149 V=150.0 PL=0
MOVL C00150 V=20.0 PL=0
MOVL C00151 V=150.0 PL=0
MOVL C00152 V=20.0 PL=0
MOVL C00153 V=150.0 PL=0
MOVL C00154 V=20.0 PL=0
MOVL C00155 V=150.0 PL=0
MOVL C00156 V=20.0 PL=0
MOVL C00157 V=150.0 PL=0
MOVL C00158 V=20.0 PL=0
MOVL C00159 V=150.0 PL=0
MOVL C00160 V=20.0 PL=0
MOVL C00161 V=150.0 PL=0
MOVL C00162 V=20.0 PL=0
MOVL C00163 V=150.0 PL=0
MOVL C00164 V=20.0 PL=0
MOVL C00165 V=20.0 PL=0
MOVL C00166 V=150.0 PL=0
MOVL C00167 V=20.0 PL=0
MOVL C00168 V=150.0 PL=0
MOVL C00169 V=20.0 PL=0
MOVL C00170 V=20.0 PL=0
MOVL C00171 V=150.0 PL=0
MOVL C00172 V=20.0 PL=0
MOVL C00173 V=150.0 PL=0
MOVL C00174 V=20.0 PL=0
MOVL C00175 V=20.0 PL=0
MOVL C00176 V=150.0 PL=0
MOVL C00177 V=20.0 PL=0
MOVL C00178 V=20.0 PL=0
MOVL C00179 V=10.0 PL=0
MOVL C00180 V=20.0 PL=0
MOVL C00181 V=150.0 PL=0
MOVL C00182 V=20.0 PL=0
MOVL C00183 V=20.0 PL=0
MOVL C00184 V=20.0 PL=0
MOVL C00185 V=20.0 PL=0
MOVL C00186 V=20.0 PL=0
MOVL C00187 V=20.0 PL=0
MOVL C00188 V=20.0 PL=0
MOVL C00189 V=20.0 PL=0
MOVL C00190 V=20.0 PL=0
MOVL C00191 V=20.0 PL=0
MOVL C00192 V=20.0 PL=0
MOVL C00193 V=20.0 PL=0
MOVL C00194 V=150.0 PL=0
MOVL C00195 V=20.0 PL=0
MOVL C00196 V=20.0 PL=0
MOVL C00197 V=20.0 PL=0
MOVL C00198 V=20.0 PL=0
MOVL C00199 V=20.0 PL=0
MOVL C00200 V=20.0 PL=0
MOVL C00201 V=20.0 PL=0
MOVL C00202 V=20.0 PL=0
MOVL C00203 V=20.0 PL=0
MOVL C00204 V=20.0 PL=0
MOVL C00205 V=20.0 PL=0
MOVL C00206 V=20.0 PL=0
MOVL C00207 V=20.0 PL=0
MOVL C00208 V=20.0 PL=0
MOVL C00209 V=20.0 PL=0
MOVL C00210 V=20.0 PL=0
MOVL C00211 V=20.0 PL=0
MOVL C00212 V=20.0 PL=0
MOVL C00213 V=20.0 PL=0
MOVL C00214 V=150.0 PL=0
MOVL C00215 V=150.0 PL=0
MOVL C00216 V=150.0 PL=0
MOVL C00217 V=150.0 PL=0
MOVL C00218 V=150.0 PL=0
MOVL C00219 V=20.0 PL=0
MOVL C00220 V=20.0 PL=0
MOVL C00221 V=20.0 PL=0
MOVL C00222 V=20.0 PL=0
MOVL C00223 V=20.0 PL=0
MOVL C00224 V=20.0 PL=0
MOVL C00225 V=20.0 PL=0
MOVL C00226 V=20.0 PL=0
MOVL C00227 V=20.0 PL=0
MOVL C00228 V=20.0 PL=0
MOVL C00229 V=20.0 PL=0
MOVL C00230 V=20.0 PL=0
MOVL C00231 V=20.0 PL=0
MOVL C00232 V=150.0 PL=0
MOVL C00233 V=150.0 PL=0
MOVL C00234 V=150.0 PL=0
MOVL C00235 V=150.0 PL=0
MOVL C00236 V=20.0 PL=0
MOVL C00237 V=20.0 PL=0
MOVL C00238 V=20.0 PL=0
MOVL C00239 V=20.0 PL=0
MOVL C00240 V=20.0 PL=0
MOVL C00241 V=20.0 PL=0
MOVL C00242 V=20.0 PL=0
MOVL C00243 V=20.0 PL=0
MOVL C00244 V=20.0 PL=0
MOVL C00245 V=20.0 PL=0
MOVL C00246 V=20.0 PL=0
MOVL C00247 V=20.0 PL=0
MOVL C00248 V=150.0 PL=0
MOVL C00249 V=20.0 PL=0
MOVL C00250 V=150.0 PL=0
MOVL C00251 V=150.0 PL=0
MOVL C00252 V=150.0 PL=0
MOVL C00253 V=150.0 PL=0
MOVL C00254 V=150.0 PL=0
MOVL C00255 V=20.0 PL=0
MOVL C00256 V=20.0 PL=0
MOVL C00257 V=20.0 PL=0
MOVL C00258 V=20.0 PL=0
MOVL C00259 V=20.0 PL=0
MOVL C00260 V=20.0 PL=0
MOVL C00261 V=20.0 PL=0
MOVL C00262 V=20.0 PL=0
MOVL C00263 V=20.0 PL=0
MOVL C00264 V=20.0 PL=0
MOVL C00265 V=20.0 PL=0
MOVL C00266 V=20.0 PL=0
MOVL C00267 V=20.0 PL=0
MOVL C00268 V=20.0 PL=0
MOVL C00269 V=20.0 PL=0
MOVL C00270 V=20.0 PL=0
MOVL C00271 V=20.0 PL=0
MOVL C00272 V=20.0 PL=0
MOVL C00273 V=20.0 PL=0
MOVL C00274 V=20.0 PL=0
MOVL C00275 V=20.0 PL=0
MOVL C00276 V=20.0 PL=0
MOVL C00277 V=20.0 PL=0
MOVL C00278 V=20.0 PL=0
MOVL C00279 V=20.0 PL=0
MOVL C00280 V=20.0 PL=0
MOVL C00281 V=20.0 PL=0
MOVL C00282 V=20.0 PL=0
MOVL C00283 V=20.0 PL=0
MOVL C00284 V=20.0 PL=0
MOVL C00285 V=20.0 PL=0
MOVL C00286 V=20.0 PL=0
MOVL C00287 V=20.0 PL=0
MOVL C00288 V=20.0 PL=0
MOVL C00289 V=20.0 PL=0
MOVL C00290 V=20.0 PL=0
MOVL C00291 V=20.0 PL=0
MOVL C00292 V=20.0 PL=0
MOVL C00293 V=20.0 PL=0
MOVL C00294 V=20.0 PL=0
MOVL C00295 V=20.0 PL=0
MOVL C00296 V=20.0 PL=0
MOVL C00297 V=20.0 PL=0
MOVL C00298 V=20.0 PL=0
MOVL C00299 V=20.0 PL=0
MOVL C00300 V=20.0 PL=0
MOVL C00301 V=20.0 PL=0
MOVL C00302 V=20.0 PL=0
MOVL C00303 V=20.0 PL=0
MOVL C00304 V=20.0 PL=0
MOVL C00305 V=20.0 PL=0
MOVL C00306 V=20.0 PL=0
MOVL C00307 V=20.0 PL=0
MOVL C00308 V=20.0 PL=0
MOVL C00309 V=20.0 PL=0
MOVL C00310 V=20.0 PL=0
MOVL C00311 V=20.0 PL=0
MOVL C00312 V=20.0 PL=0
MOVL C00313 V=20.0 PL=0
MOVL C00314 V=20.0 PL=0
MOVL C00315 V=20.0 PL=0
MOVL C00316 V=20.0 PL=0
MOVL C00317 V=20.0 PL=0
MOVL C00318 V=20.0 PL=0
MOVL C00319 V=20.0 PL=0
MOVL C00320 V=20.0 PL=0
MOVL C00321 V=20.0 PL=0
MOVL C00322 V=20.0 PL=0
MOVL C00323 V=20.0 PL=0
MOVL C00324 V=20.0 PL=0
MOVL C00325 V=20.0 PL=0
MOVL C00326 V=20.0 PL=0
MOVL C00327 V=20.0 PL=0
MOVL C00328 V=20.0 PL=0
MOVL C00329 V=20.0 PL=0
MOVL C00330 V=20.0 PL=0
MOVL C00331 V=20.0 PL=0
MOVL C00332 V=20.0 PL=0
MOVL C00333 V=20.0 PL=0
MOVL C00334 V=20.0 PL=0
MOVL C00335 V=20.0 PL=0
MOVL C00336 V=20.0 PL=0
MOVL C00337 V=20.0 PL=0
MOVL C00338 V=20.0 PL=0
MOVL C00339 V=20.0 PL=0
MOVL C00340 V=20.0 PL=0
MOVL C00341 V=20.0 PL=0
MOVL C00342 V=20.0 PL=0
MOVL C00343 V=20.0 PL=0
MOVL C00344 V=20.0 PL=0
MOVL C00345 V=20.0 PL=0
